Yaskawa INFORM job: aprem2TRJ4.JBI

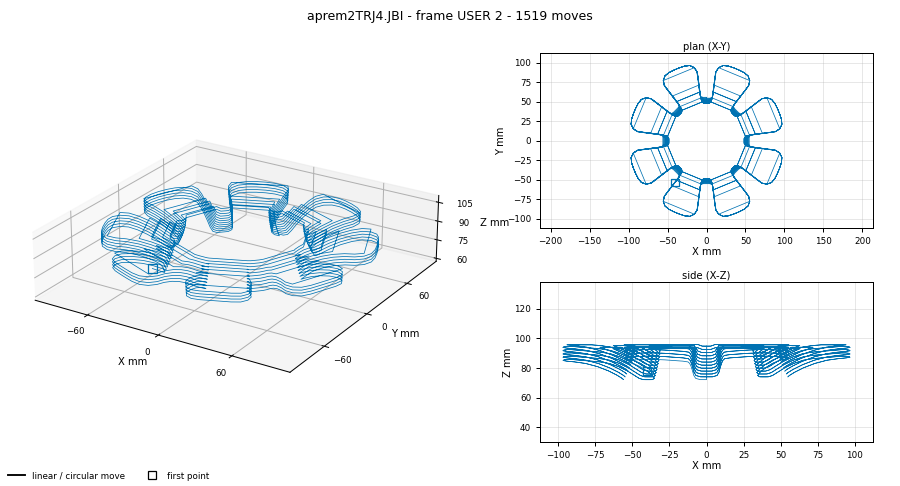
[picture p0: tool path of aprem2TRJ4.JBI in frame USER 2, 1519 of 1519 moves have a stored position in this frame; points joined in program order, loops and branches not executed]
/JOB
//NAME aprem2TRJ4
//POS
///NPOS 1519,0,1519,0,0,0
///USER 2
///TOOL 1
///POSTYPE USER
///RECTAN
///RCONF 1,0,0,0,0,0,0,0,0,0,0,0,0,0,0,0,0,0,0,0,0,0,0,0
C00000=-40.007,-53.324,78.036,177.7295,-3.1005,0.0000
C00001=-36.517,-48.718,75.143,178.8242,-1.7083,0.0000
C00002=-35.037,-45.351,73.015,-179.8825,17.3486,0.0000
C00003=-36.538,-42.505,72.166,160.0580,24.5520,0.0000
C00004=-38.303,-40.803,72.129,156.0408,22.3844,0.0000
C00005=-39.567,-39.567,72.154,156.8171,23.1818,0.0000
C00006=-40.803,-38.303,72.129,157.6162,23.9597,0.0000
C00007=-42.506,-36.538,72.166,155.4471,19.9396,0.0000
C00008=-45.352,-35.037,73.015,162.6519,-0.1179,0.0000
C00009=-48.718,-36.517,75.143,-178.2917,1.1758,0.0000
C00010=-53.324,-40.007,78.036,-176.8995,2.2705,0.0000
C00011=-59.196,-44.618,80.927,-176.4745,2.6327,0.0000
C00012=-65.578,-49.604,83.062,-176.2466,2.8111,0.0000
C00013=-71.524,-53.949,84.088,-176.0077,2.0393,0.0000
C00014=-77.795,-55.184,84.621,-177.1914,-0.2563,0.0000
C00015=-83.601,-53.037,85.050,-178.9039,-0.7847,0.0000
C00016=-87.741,-47.957,85.481,-179.9577,-0.0772,0.0000
C00017=-90.934,-41.602,85.762,-179.9958,-0.0092,0.0000
C00018=-93.717,-34.883,85.762,-179.9965,-0.0095,0.0000
C00019=-95.953,-28.131,85.481,-179.9754,-0.0845,0.0000
C00020=-96.617,-21.612,85.050,179.7797,-1.3299,0.0000
C00021=-94.030,-15.989,84.621,178.1943,-2.1678,0.0000
C00022=-88.723,-12.427,84.088,175.7377,-1.3847,0.0000
C00023=-81.446,-11.295,83.062,175.3629,-0.6685,0.0000
C00024=-73.408,-10.308,80.927,175.6494,-0.6331,0.0000
C00025=-65.995,-9.417,78.036,176.2047,-0.5882,0.0000
C00026=-60.270,-8.627,75.143,177.9610,-0.3768,0.0000
C00027=-56.844,-7.293,73.015,-167.4643,12.3773,0.0000
C00028=-55.892,-4.219,72.166,-176.1973,30.0956,0.0000
C00029=-55.936,-1.768,72.129,178.6826,31.1925,0.0000
C00030=-55.957,0.000,72.154,179.9991,31.1998,0.0000
C00031=-55.936,1.767,72.129,-178.6816,31.1926,0.0000
C00032=-55.892,4.220,72.166,176.1946,30.0948,0.0000
C00033=-56.844,7.293,73.015,167.4645,12.3766,0.0000
C00034=-60.270,8.627,75.143,-177.9610,-0.3768,0.0000
C00035=-65.995,9.417,78.036,-176.2047,-0.5882,0.0000
C00036=-73.408,10.308,80.927,-175.6494,-0.6331,0.0000
C00037=-81.446,11.295,83.062,-175.3629,-0.6685,0.0000
C00038=-88.723,12.427,84.088,-175.7377,-1.3847,0.0000
C00039=-94.030,15.989,84.621,-178.1943,-2.1678,0.0000
C00040=-96.617,21.612,85.050,-179.7797,-1.3299,0.0000
C00041=-95.953,28.131,85.481,179.9754,-0.0845,0.0000
C00042=-93.717,34.883,85.762,179.9965,-0.0095,0.0000
C00043=-90.934,41.602,85.762,179.9958,-0.0092,0.0000
C00044=-87.741,47.957,85.481,179.9577,-0.0772,0.0000
C00045=-83.601,53.037,85.050,178.9039,-0.7847,0.0000
C00046=-77.795,55.184,84.621,177.1914,-0.2563,0.0000
C00047=-71.524,53.949,84.088,176.0077,2.0393,0.0000
C00048=-65.578,49.604,83.062,176.2466,2.8111,0.0000
C00049=-59.196,44.618,80.927,176.4745,2.6327,0.0000
C00050=-53.324,40.007,78.036,176.8995,2.2705,0.0000
C00051=-48.718,36.517,75.143,178.2917,1.1758,0.0000
C00052=-45.351,35.037,73.015,-162.6514,-0.1175,0.0000
C00053=-42.505,36.538,72.166,-155.4480,19.9420,0.0000
C00054=-40.803,38.303,72.129,-157.6156,23.9592,0.0000
C00055=-39.567,39.567,72.154,-156.8182,23.1829,0.0000
C00056=-38.303,40.803,72.129,-156.0403,22.3838,0.0000
C00057=-36.538,42.506,72.166,-160.0604,24.5529,0.0000
C00058=-35.037,45.352,73.015,179.8821,17.3481,0.0000
C00059=-36.517,48.718,75.143,-178.8242,-1.7083,0.0000
C00060=-40.007,53.324,78.036,-177.7295,-3.1005,0.0000
C00061=-44.618,59.196,80.927,-177.3673,-3.5255,0.0000
C00062=-49.604,65.578,83.062,-177.1889,-3.7534,0.0000
C00063=-53.949,71.524,84.088,-177.9607,-3.9923,0.0000
C00064=-55.184,77.795,84.621,179.7437,-2.8086,0.0000
C00065=-53.037,83.601,85.050,179.2153,-1.0961,0.0000
C00066=-47.957,87.741,85.481,179.9228,-0.0423,0.0000
C00067=-41.602,90.934,85.762,179.9908,-0.0042,0.0000
C00068=-34.883,93.717,85.762,179.9905,-0.0035,0.0000
C00069=-28.131,95.953,85.481,179.9155,-0.0246,0.0000
C00070=-21.612,96.617,85.050,178.6701,0.2203,0.0000
C00071=-15.989,94.030,84.621,177.8322,1.8057,0.0000
C00072=-12.427,88.723,84.088,178.6153,4.2623,0.0000
C00073=-11.295,81.446,83.062,179.3315,4.6371,0.0000
C00074=-10.308,73.408,80.927,179.3669,4.3506,0.0000
C00075=-9.417,65.995,78.036,179.4118,3.7953,0.0000
C00076=-8.627,60.270,75.143,179.6232,2.0390,0.0000
C00077=-7.293,56.844,73.015,-167.6234,-12.5355,0.0000
C00078=-4.220,55.892,72.166,-149.9052,-3.8054,0.0000
C00079=-1.767,55.936,72.129,-148.8074,1.3184,0.0000
C00080=0.000,55.957,72.154,-148.8002,-0.0009,0.0000
C00081=0.000,54.840,74.049,-150.2606,-0.0009,0.0000
C00082=1.666,54.823,74.024,-150.2652,-1.1897,0.0000
C00083=4.048,54.790,74.062,-151.4249,3.8705,0.0000
C00084=7.088,55.804,74.943,-168.9167,11.6638,0.0000
C00085=8.393,59.388,77.145,179.6271,-2.1340,0.0000
C00086=9.180,65.335,80.122,179.4707,-3.5331,0.0000
C00087=10.089,72.980,83.074,179.4510,-3.8704,0.0000
C00088=11.094,81.206,85.240,179.4410,-3.9838,0.0000
C00089=12.226,88.613,86.276,178.8532,-3.5972,0.0000
C00090=15.808,94.009,86.813,178.1980,-1.5172,0.0000
C00091=21.475,96.642,87.246,178.9013,-0.1852,0.0000
C00092=28.048,95.980,87.679,179.9308,0.0202,0.0000
C00093=34.856,93.728,87.962,179.9923,0.0029,0.0000
C00094=41.629,90.922,87.962,179.9925,0.0034,0.0000
C00095=48.035,87.701,87.679,179.9368,0.0347,0.0000
C00096=53.151,83.521,87.246,179.3540,0.9079,0.0000
C00097=55.296,77.652,86.813,179.7985,2.3464,0.0000
C00098=54.014,71.304,86.276,-178.2646,3.3541,0.0000
C00099=49.577,65.266,85.240,-177.5752,3.2135,0.0000
C00100=44.470,58.738,83.074,-177.6486,3.1261,0.0000
C00101=39.708,52.690,80.122,-177.8738,2.8733,0.0000
C00102=36.059,47.928,77.145,-178.7542,1.7728,0.0000
C00103=34.447,44.472,74.943,179.5730,-15.8802,0.0000
C00104=35.880,41.605,74.062,-161.3614,-23.4111,0.0000
C00105=37.588,39.944,74.024,-157.2868,-21.2665,0.0000
C00106=38.778,38.778,74.049,-158.0022,-21.9968,0.0000
C00107=39.943,37.588,74.024,-158.7340,-22.7138,0.0000
C00108=41.605,35.880,74.062,-156.5881,-18.6363,0.0000
C00109=44.472,34.447,74.943,-164.1205,0.4274,0.0000
C00110=47.928,36.059,77.145,178.2272,-1.2458,0.0000
C00111=52.690,39.708,80.122,177.1267,-2.1262,0.0000
C00112=58.738,44.470,83.074,176.8739,-2.3514,0.0000
C00113=65.266,49.577,85.240,176.7865,-2.4248,0.0000
C00114=71.304,54.014,86.276,176.6459,-1.7354,0.0000
C00115=77.652,55.296,86.813,177.6536,0.2015,0.0000
C00116=83.521,53.151,87.246,179.0921,0.6460,0.0000
C00117=87.701,48.035,87.679,179.9653,0.0632,0.0000
C00118=90.922,41.629,87.962,179.9966,0.0075,0.0000
C00119=93.728,34.856,87.962,179.9971,0.0077,0.0000
C00120=95.980,28.048,87.679,179.9798,0.0692,0.0000
C00121=96.642,21.475,87.246,-179.8148,1.0987,0.0000
C00122=94.009,15.808,86.813,-178.4828,1.8020,0.0000
C00123=88.613,12.226,86.276,-176.4028,1.1468,0.0000
C00124=81.206,11.094,85.240,-176.0162,0.5590,0.0000
C00125=72.980,10.089,83.074,-176.1296,0.5490,0.0000
C00126=65.335,9.180,80.122,-176.4669,0.5293,0.0000
C00127=59.388,8.393,77.145,-177.8660,0.3729,0.0000
C00128=55.804,7.088,74.943,168.3362,-11.0833,0.0000
C00129=54.790,4.048,74.062,176.1295,-28.5751,0.0000
C00130=54.823,1.666,74.024,-178.8103,-29.7348,0.0000
C00131=54.840,0.000,74.049,-179.9991,-29.7394,0.0000
C00132=54.823,-1.665,74.024,178.8094,-29.7348,0.0000
C00133=54.790,-4.048,74.062,-176.1270,-28.5741,0.0000
C00134=55.804,-7.088,74.943,-168.3364,-11.0826,0.0000
C00135=59.388,-8.393,77.145,177.8660,0.3729,0.0000
C00136=65.335,-9.180,80.122,176.4669,0.5293,0.0000
C00137=72.980,-10.089,83.074,176.1296,0.5490,0.0000
C00138=81.206,-11.094,85.240,176.0162,0.5590,0.0000
C00139=88.613,-12.226,86.276,176.4028,1.1468,0.0000
C00140=94.009,-15.808,86.813,178.4828,1.8020,0.0000
C00141=96.642,-21.475,87.246,179.8148,1.0987,0.0000
C00142=95.980,-28.048,87.679,-179.9798,0.0692,0.0000
C00143=93.728,-34.856,87.962,-179.9971,0.0077,0.0000
C00144=90.922,-41.629,87.962,-179.9966,0.0075,0.0000
C00145=87.701,-48.035,87.679,-179.9653,0.0632,0.0000
C00146=83.521,-53.151,87.246,-179.0921,0.6460,0.0000
C00147=77.652,-55.296,86.813,-177.6536,0.2015,0.0000
C00148=71.304,-54.014,86.276,-176.6459,-1.7354,0.0000
C00149=65.266,-49.577,85.240,-176.7865,-2.4248,0.0000
C00150=58.738,-44.470,83.074,-176.8739,-2.3514,0.0000
C00151=52.690,-39.708,80.122,-177.1267,-2.1262,0.0000
C00152=47.928,-36.059,77.145,-178.2272,-1.2458,0.0000
C00153=44.472,-34.447,74.943,164.1198,0.4270,0.0000
C00154=41.605,-35.880,74.062,156.5889,-18.6386,0.0000
C00155=39.944,-37.588,74.024,158.7335,-22.7132,0.0000
C00156=38.778,-38.778,74.049,158.0032,-21.9978,0.0000
C00157=37.588,-39.943,74.024,157.2862,-21.2660,0.0000
C00158=35.880,-41.605,74.062,161.3637,-23.4119,0.0000
C00159=34.447,-44.472,74.943,-179.5726,-15.8795,0.0000
C00160=36.059,-47.928,77.145,178.7542,1.7728,0.0000
C00161=39.708,-52.690,80.122,177.8738,2.8733,0.0000
C00162=44.470,-58.738,83.074,177.6486,3.1261,0.0000
C00163=49.577,-65.266,85.240,177.5752,3.2135,0.0000
C00164=54.014,-71.304,86.276,178.2646,3.3541,0.0000
C00165=55.296,-77.652,86.813,-179.7985,2.3464,0.0000
C00166=53.151,-83.521,87.246,-179.3540,0.9079,0.0000
C00167=48.035,-87.701,87.679,-179.9368,0.0347,0.0000
C00168=41.629,-90.922,87.962,-179.9925,0.0034,0.0000
C00169=34.856,-93.728,87.962,-179.9923,0.0029,0.0000
C00170=28.048,-95.980,87.679,-179.9308,0.0202,0.0000
C00171=21.475,-96.642,87.246,-178.9013,-0.1852,0.0000
C00172=15.808,-94.009,86.813,-178.1980,-1.5172,0.0000
C00173=12.226,-88.613,86.276,-178.8532,-3.5972,0.0000
C00174=11.094,-81.206,85.240,-179.4410,-3.9838,0.0000
C00175=10.089,-72.980,83.074,-179.4510,-3.8704,0.0000
C00176=9.180,-65.335,80.122,-179.4707,-3.5331,0.0000
C00177=8.393,-59.388,77.145,-179.6271,-2.1340,0.0000
C00178=7.088,-55.804,74.943,168.9167,11.6638,0.0000
C00179=4.048,-54.790,74.062,151.4249,3.8705,0.0000
C00180=1.666,-54.823,74.024,150.2652,-1.1897,0.0000
C00181=0.000,-54.840,74.049,150.2606,-0.0009,0.0000
C00182=0.000,-54.840,74.049,150.2606,-0.0009,0.0000
C00183=-1.665,-54.823,74.024,150.2652,1.1906,0.0000
C00184=-4.048,-54.790,74.062,151.4259,-3.8730,0.0000
C00185=-7.088,-55.804,74.943,168.9174,-11.6636,0.0000
C00186=-8.393,-59.388,77.145,-179.6271,2.1340,0.0000
C00187=-9.180,-65.335,80.122,-179.4707,3.5331,0.0000
C00188=-10.089,-72.980,83.074,-179.4510,3.8704,0.0000
C00189=-11.094,-81.206,85.240,-179.4410,3.9838,0.0000
C00190=-12.226,-88.613,86.276,-178.8532,3.5972,0.0000
C00191=-15.808,-94.009,86.813,-178.1980,1.5172,0.0000
C00192=-21.475,-96.642,87.246,-178.9013,0.1852,0.0000
C00193=-28.048,-95.980,87.679,-179.9308,-0.0202,0.0000
C00194=-34.856,-93.728,87.962,-179.9923,-0.0029,0.0000
C00195=-41.629,-90.922,87.962,-179.9925,-0.0034,0.0000
C00196=-48.035,-87.701,87.679,-179.9368,-0.0347,0.0000
C00197=-53.151,-83.521,87.246,-179.3540,-0.9079,0.0000
C00198=-55.296,-77.652,86.813,-179.7985,-2.3464,0.0000
C00199=-54.014,-71.304,86.276,178.2646,-3.3541,0.0000
C00200=-49.577,-65.266,85.240,177.5752,-3.2135,0.0000
C00201=-44.470,-58.738,83.074,177.6486,-3.1261,0.0000
C00202=-39.708,-52.690,80.122,177.8738,-2.8733,0.0000
C00203=-36.059,-47.928,77.145,178.7542,-1.7728,0.0000
C00204=-34.447,-44.472,74.943,-179.5730,15.8802,0.0000
C00205=-35.880,-41.605,74.062,161.3614,23.4111,0.0000
C00206=-37.588,-39.944,74.024,157.2868,21.2665,0.0000
C00207=-38.778,-38.778,74.049,158.0022,21.9968,0.0000
C00208=-39.943,-37.588,74.024,158.7340,22.7138,0.0000
C00209=-41.605,-35.880,74.062,156.5881,18.6363,0.0000
C00210=-44.472,-34.447,74.943,164.1205,-0.4274,0.0000
C00211=-47.928,-36.059,77.145,-178.2272,1.2458,0.0000
C00212=-52.690,-39.708,80.122,-177.1267,2.1262,0.0000
C00213=-58.738,-44.470,83.074,-176.8739,2.3514,0.0000
C00214=-65.266,-49.577,85.240,-176.7865,2.4248,0.0000
C00215=-71.304,-54.014,86.276,-176.6459,1.7354,0.0000
C00216=-77.652,-55.296,86.813,-177.6536,-0.2015,0.0000
C00217=-83.521,-53.151,87.246,-179.0921,-0.6460,0.0000
C00218=-87.701,-48.035,87.679,-179.9653,-0.0632,0.0000
C00219=-90.922,-41.629,87.962,-179.9966,-0.0075,0.0000
C00220=-93.728,-34.856,87.962,-179.9971,-0.0077,0.0000
C00221=-95.980,-28.048,87.679,-179.9798,-0.0692,0.0000
C00222=-96.642,-21.475,87.246,179.8148,-1.0987,0.0000
C00223=-94.009,-15.808,86.813,178.4828,-1.8020,0.0000
C00224=-88.613,-12.226,86.276,176.4028,-1.1468,0.0000
C00225=-81.206,-11.094,85.240,176.0162,-0.5590,0.0000
C00226=-72.980,-10.089,83.074,176.1296,-0.5490,0.0000
C00227=-65.335,-9.180,80.122,176.4669,-0.5293,0.0000
C00228=-59.388,-8.393,77.145,177.8660,-0.3729,0.0000
C00229=-55.804,-7.088,74.943,-168.3362,11.0833,0.0000
C00230=-54.790,-4.048,74.062,-176.1295,28.5751,0.0000
C00231=-54.823,-1.666,74.024,178.8103,29.7348,0.0000
C00232=-54.840,0.000,74.049,179.9991,29.7394,0.0000
C00233=-54.823,1.665,74.024,-178.8094,29.7348,0.0000
C00234=-54.790,4.048,74.062,176.1270,28.5741,0.0000
C00235=-55.804,7.088,74.943,168.3364,11.0826,0.0000
C00236=-59.388,8.393,77.145,-177.8660,-0.3729,0.0000
C00237=-65.335,9.180,80.122,-176.4669,-0.5293,0.0000
C00238=-72.980,10.089,83.074,-176.1296,-0.5490,0.0000
C00239=-81.206,11.094,85.240,-176.0162,-0.5590,0.0000
C00240=-88.613,12.226,86.276,-176.4028,-1.1468,0.0000
C00241=-94.009,15.808,86.813,-178.4828,-1.8020,0.0000
C00242=-96.642,21.475,87.246,-179.8148,-1.0987,0.0000
C00243=-95.980,28.048,87.679,179.9798,-0.0692,0.0000
C00244=-93.728,34.856,87.962,179.9971,-0.0077,0.0000
C00245=-90.922,41.629,87.962,179.9966,-0.0075,0.0000
C00246=-87.701,48.035,87.679,179.9653,-0.0632,0.0000
C00247=-83.521,53.151,87.246,179.0921,-0.6460,0.0000
C00248=-77.652,55.296,86.813,177.6536,-0.2015,0.0000
C00249=-71.304,54.014,86.276,176.6459,1.7354,0.0000
C00250=-65.266,49.577,85.240,176.7865,2.4248,0.0000
C00251=-58.738,44.470,83.074,176.8739,2.3514,0.0000
C00252=-52.690,39.708,80.122,177.1267,2.1262,0.0000
C00253=-47.928,36.059,77.145,178.2272,1.2458,0.0000
C00254=-44.472,34.447,74.943,-164.1198,-0.4270,0.0000
C00255=-41.605,35.880,74.062,-156.5889,18.6386,0.0000
C00256=-39.944,37.588,74.024,-158.7335,22.7132,0.0000
C00257=-38.778,38.778,74.049,-158.0032,21.9978,0.0000
C00258=-37.588,39.943,74.024,-157.2862,21.2660,0.0000
C00259=-35.880,41.605,74.062,-161.3637,23.4119,0.0000
C00260=-34.447,44.472,74.943,179.5726,15.8795,0.0000
C00261=-36.059,47.928,77.145,-178.7542,-1.7728,0.0000
C00262=-39.708,52.690,80.122,-177.8738,-2.8733,0.0000
C00263=-44.470,58.738,83.074,-177.6486,-3.1261,0.0000
C00264=-49.577,65.266,85.240,-177.5752,-3.2135,0.0000
C00265=-54.014,71.304,86.276,-178.2646,-3.3541,0.0000
C00266=-55.296,77.652,86.813,179.7985,-2.3464,0.0000
C00267=-53.151,83.521,87.246,179.3540,-0.9079,0.0000
C00268=-48.035,87.701,87.679,179.9368,-0.0347,0.0000
C00269=-41.629,90.922,87.962,179.9925,-0.0034,0.0000
C00270=-34.856,93.728,87.962,179.9923,-0.0029,0.0000
C00271=-28.048,95.980,87.679,179.9308,-0.0202,0.0000
C00272=-21.475,96.642,87.246,178.9013,0.1852,0.0000
C00273=-15.808,94.009,86.813,178.1980,1.5172,0.0000
C00274=-12.226,88.613,86.276,178.8532,3.5972,0.0000
C00275=-11.094,81.206,85.240,179.4410,3.9838,0.0000
C00276=-10.089,72.980,83.074,179.4510,3.8704,0.0000
C00277=-9.180,65.335,80.122,179.4707,3.5331,0.0000
C00278=-8.393,59.388,77.145,179.6271,2.1340,0.0000
C00279=-7.088,55.804,74.943,-168.9174,-11.6636,0.0000
C00280=-4.048,54.790,74.062,-151.4259,-3.8730,0.0000
C00281=-1.665,54.823,74.024,-150.2652,1.1906,0.0000
C00282=0.000,54.840,74.049,-150.2606,-0.0009,0.0000
C00283=0.000,53.776,75.975,-151.9017,-0.0008,0.0000
C00284=1.568,53.762,75.948,-151.9034,-1.0593,0.0000
C00285=3.884,53.739,75.988,-153.1148,3.8750,0.0000
C00286=6.894,54.818,76.900,-170.1649,10.7294,0.0000
C00287=8.175,58.565,79.173,179.6434,-2.1517,0.0000
C00288=8.965,64.737,82.228,179.5331,-3.2135,0.0000
C00289=9.898,72.606,85.234,179.5371,-3.3364,0.0000
C00290=10.924,81.005,87.424,179.5509,-3.2738,0.0000
C00291=12.061,88.524,88.468,179.0976,-2.8742,0.0000
C00292=15.662,93.991,89.008,178.5900,-1.1973,0.0000
C00293=21.365,96.662,89.443,179.1515,-0.1450,0.0000
C00294=27.983,96.002,89.878,179.9474,0.0153,0.0000
C00295=34.834,93.736,90.162,179.9942,0.0022,0.0000
C00296=41.650,90.913,90.162,179.9944,0.0026,0.0000
C00297=48.097,87.670,89.878,179.9520,0.0264,0.0000
C00298=53.243,83.458,89.443,179.5025,0.7025,0.0000
C00299=55.387,77.537,89.008,179.8495,1.8433,0.0000
C00300=54.067,71.124,88.468,-178.6043,2.6703,0.0000
C00301=49.554,65.004,87.424,-178.0010,2.6331,0.0000
C00302=44.341,58.339,85.234,-177.9664,2.6872,0.0000
C00303=39.437,52.115,82.228,-178.0562,2.6030,0.0000
C00304=35.631,47.192,79.173,-178.7302,1.7738,0.0000
C00305=33.888,43.637,76.900,179.3468,-14.3899,0.0000
C00306=35.253,40.746,75.988,-162.7447,-22.1169,0.0000
C00307=36.906,39.124,75.948,-158.6653,-20.0234,0.0000
C00308=38.025,38.025,75.975,-159.3164,-20.6826,0.0000
C00309=39.124,36.906,75.948,-159.9771,-21.3352,0.0000
C00310=40.746,35.253,75.988,-157.8823,-17.2529,0.0000
C00311=43.637,33.888,76.901,-165.6107,0.6536,0.0000
C00312=47.192,35.631,79.173,178.2262,-1.2698,0.0000
C00313=52.115,39.437,82.228,177.3970,-1.9438,0.0000
C00314=58.339,44.341,85.234,177.3128,-2.0336,0.0000
C00315=65.004,49.554,87.424,177.3669,-1.9990,0.0000
C00316=71.124,54.067,88.468,177.3297,-1.3957,0.0000
C00317=77.537,55.387,89.008,178.1567,0.1505,0.0000
C00318=83.458,53.243,89.443,179.2975,0.4975,0.0000
C00319=87.670,48.097,89.878,179.9736,0.0480,0.0000
C00320=90.913,41.650,90.162,179.9974,0.0056,0.0000
C00321=93.736,34.834,90.162,179.9978,0.0058,0.0000
C00322=96.002,27.983,89.878,179.9847,0.0526,0.0000
C00323=96.662,21.365,89.443,-179.8550,0.8485,0.0000
C00324=93.991,15.662,89.008,-178.8027,1.4100,0.0000
C00325=88.524,12.061,88.468,-177.1258,0.9024,0.0000
C00326=81.005,10.924,87.424,-176.7262,0.4491,0.0000
C00327=72.606,9.898,85.234,-176.6636,0.4629,0.0000
C00328=64.737,8.965,82.228,-176.7865,0.4669,0.0000
C00329=58.565,8.175,79.173,-177.8483,0.3566,0.0000
C00330=54.818,6.894,76.900,169.2706,-9.8351,0.0000
C00331=53.739,3.884,75.988,176.1250,-26.8852,0.0000
C00332=53.762,1.568,75.948,-178.9407,-28.0966,0.0000
C00333=53.776,0.000,75.975,-179.9992,-28.0983,0.0000
C00334=53.762,-1.568,75.948,178.9399,-28.0967,0.0000
C00335=53.739,-3.885,75.988,-176.1225,-26.8842,0.0000
C00336=54.819,-6.894,76.901,-169.2709,-9.8343,0.0000
C00337=58.565,-8.175,79.173,177.8483,0.3566,0.0000
C00338=64.737,-8.965,82.228,176.7865,0.4669,0.0000
C00339=72.606,-9.898,85.234,176.6636,0.4629,0.0000
C00340=81.005,-10.924,87.424,176.7262,0.4491,0.0000
C00341=88.524,-12.061,88.468,177.1258,0.9024,0.0000
C00342=93.991,-15.662,89.008,178.8027,1.4100,0.0000
C00343=96.662,-21.365,89.443,179.8550,0.8485,0.0000
C00344=96.002,-27.983,89.878,-179.9847,0.0526,0.0000
C00345=93.736,-34.834,90.162,-179.9978,0.0058,0.0000
C00346=90.913,-41.650,90.162,-179.9974,0.0056,0.0000
C00347=87.670,-48.097,89.878,-179.9736,0.0480,0.0000
C00348=83.458,-53.243,89.443,-179.2975,0.4975,0.0000
C00349=77.537,-55.387,89.008,-178.1567,0.1505,0.0000
C00350=71.124,-54.067,88.468,-177.3297,-1.3957,0.0000
C00351=65.004,-49.554,87.424,-177.3669,-1.9990,0.0000
C00352=58.339,-44.341,85.234,-177.3128,-2.0336,0.0000
C00353=52.115,-39.437,82.228,-177.3970,-1.9438,0.0000
C00354=47.192,-35.631,79.173,-178.2262,-1.2698,0.0000
C00355=43.637,-33.888,76.900,165.6101,0.6532,0.0000
C00356=40.746,-35.253,75.988,157.8831,-17.2553,0.0000
C00357=39.124,-36.906,75.948,159.9766,-21.3347,0.0000
C00358=38.025,-38.025,75.975,159.3174,-20.6836,0.0000
C00359=36.906,-39.124,75.948,158.6648,-20.0229,0.0000
C00360=35.253,-40.746,75.988,162.7471,-22.1177,0.0000
C00361=33.888,-43.637,76.901,-179.3464,-14.3893,0.0000
C00362=35.631,-47.192,79.173,178.7302,1.7738,0.0000
C00363=39.437,-52.115,82.228,178.0562,2.6030,0.0000
C00364=44.341,-58.339,85.234,177.9664,2.6872,0.0000
C00365=49.554,-65.004,87.424,178.0010,2.6331,0.0000
C00366=54.067,-71.124,88.468,178.6043,2.6703,0.0000
C00367=55.387,-77.537,89.008,-179.8495,1.8433,0.0000
C00368=53.243,-83.458,89.443,-179.5025,0.7025,0.0000
C00369=48.097,-87.670,89.878,-179.9520,0.0264,0.0000
C00370=41.650,-90.913,90.162,-179.9944,0.0026,0.0000
C00371=34.834,-93.736,90.162,-179.9942,0.0022,0.0000
C00372=27.983,-96.002,89.878,-179.9474,0.0153,0.0000
C00373=21.365,-96.662,89.443,-179.1515,-0.1450,0.0000
C00374=15.662,-93.991,89.008,-178.5900,-1.1973,0.0000
C00375=12.061,-88.524,88.468,-179.0976,-2.8742,0.0000
C00376=10.924,-81.005,87.424,-179.5509,-3.2738,0.0000
C00377=9.898,-72.606,85.234,-179.5371,-3.3364,0.0000
C00378=8.965,-64.737,82.228,-179.5331,-3.2135,0.0000
C00379=8.175,-58.565,79.173,-179.6434,-2.1517,0.0000
C00380=6.894,-54.818,76.900,170.1649,10.7294,0.0000
C00381=3.884,-53.739,75.988,153.1148,3.8750,0.0000
C00382=1.568,-53.762,75.948,151.9034,-1.0593,0.0000
C00383=0.000,-53.776,75.975,151.9017,-0.0008,0.0000
C00384=0.000,-53.776,75.975,151.9017,-0.0008,0.0000
C00385=-1.568,-53.762,75.948,151.9033,1.0601,0.0000
C00386=-3.885,-53.739,75.988,153.1158,-3.8775,0.0000
C00387=-6.894,-54.819,76.901,170.1657,-10.7291,0.0000
C00388=-8.175,-58.565,79.173,-179.6434,2.1517,0.0000
C00389=-8.965,-64.737,82.228,-179.5331,3.2135,0.0000
C00390=-9.898,-72.606,85.234,-179.5371,3.3364,0.0000
C00391=-10.924,-81.005,87.424,-179.5509,3.2738,0.0000
C00392=-12.061,-88.524,88.468,-179.0976,2.8742,0.0000
C00393=-15.662,-93.991,89.008,-178.5900,1.1973,0.0000
C00394=-21.365,-96.662,89.443,-179.1515,0.1450,0.0000
C00395=-27.983,-96.002,89.878,-179.9474,-0.0153,0.0000
C00396=-34.834,-93.736,90.162,-179.9942,-0.0022,0.0000
C00397=-41.650,-90.913,90.162,-179.9944,-0.0026,0.0000
C00398=-48.097,-87.670,89.878,-179.9520,-0.0264,0.0000
C00399=-53.243,-83.458,89.443,-179.5025,-0.7025,0.0000
C00400=-55.387,-77.537,89.008,-179.8495,-1.8433,0.0000
C00401=-54.067,-71.124,88.468,178.6043,-2.6703,0.0000
C00402=-49.554,-65.004,87.424,178.0010,-2.6331,0.0000
C00403=-44.341,-58.339,85.234,177.9664,-2.6872,0.0000
C00404=-39.437,-52.115,82.228,178.0562,-2.6030,0.0000
C00405=-35.631,-47.192,79.173,178.7302,-1.7738,0.0000
C00406=-33.888,-43.637,76.900,-179.3468,14.3899,0.0000
C00407=-35.253,-40.746,75.988,162.7447,22.1169,0.0000
C00408=-36.906,-39.124,75.948,158.6653,20.0234,0.0000
C00409=-38.025,-38.025,75.975,159.3164,20.6826,0.0000
C00410=-39.124,-36.906,75.948,159.9771,21.3352,0.0000
C00411=-40.746,-35.253,75.988,157.8823,17.2529,0.0000
C00412=-43.637,-33.888,76.901,165.6107,-0.6536,0.0000
C00413=-47.192,-35.631,79.173,-178.2262,1.2698,0.0000
C00414=-52.115,-39.437,82.228,-177.3970,1.9438,0.0000
C00415=-58.339,-44.341,85.234,-177.3128,2.0336,0.0000
C00416=-65.004,-49.554,87.424,-177.3669,1.9990,0.0000
C00417=-71.124,-54.067,88.468,-177.3297,1.3957,0.0000
C00418=-77.537,-55.387,89.008,-178.1567,-0.1505,0.0000
C00419=-83.458,-53.243,89.443,-179.2975,-0.4975,0.0000
C00420=-87.670,-48.097,89.878,-179.9736,-0.0480,0.0000
C00421=-90.913,-41.650,90.162,-179.9974,-0.0056,0.0000
C00422=-93.736,-34.834,90.162,-179.9978,-0.0058,0.0000
C00423=-96.002,-27.983,89.878,-179.9847,-0.0526,0.0000
C00424=-96.662,-21.365,89.443,179.8550,-0.8485,0.0000
C00425=-93.991,-15.662,89.008,178.8027,-1.4100,0.0000
C00426=-88.524,-12.061,88.468,177.1258,-0.9024,0.0000
C00427=-81.005,-10.924,87.424,176.7262,-0.4491,0.0000
C00428=-72.606,-9.898,85.234,176.6636,-0.4629,0.0000
C00429=-64.737,-8.965,82.228,176.7865,-0.4669,0.0000
C00430=-58.565,-8.175,79.173,177.8483,-0.3566,0.0000
C00431=-54.818,-6.894,76.900,-169.2706,9.8351,0.0000
C00432=-53.739,-3.884,75.988,-176.1250,26.8852,0.0000
C00433=-53.762,-1.568,75.948,178.9407,28.0966,0.0000
C00434=-53.776,0.000,75.975,179.9992,28.0983,0.0000
C00435=-53.762,1.568,75.948,-178.9399,28.0967,0.0000
C00436=-53.739,3.885,75.988,176.1225,26.8842,0.0000
C00437=-54.819,6.894,76.901,169.2709,9.8343,0.0000
C00438=-58.565,8.175,79.173,-177.8483,-0.3566,0.0000
C00439=-64.737,8.965,82.228,-176.7865,-0.4669,0.0000
C00440=-72.606,9.898,85.234,-176.6636,-0.4629,0.0000
C00441=-81.005,10.924,87.424,-176.7262,-0.4491,0.0000
C00442=-88.524,12.061,88.468,-177.1258,-0.9024,0.0000
C00443=-93.991,15.662,89.008,-178.8027,-1.4100,0.0000
C00444=-96.662,21.365,89.443,-179.8550,-0.8485,0.0000
C00445=-96.002,27.983,89.878,179.9847,-0.0526,0.0000
C00446=-93.736,34.834,90.162,179.9978,-0.0058,0.0000
C00447=-90.913,41.650,90.162,179.9974,-0.0056,0.0000
C00448=-87.670,48.097,89.878,179.9736,-0.0480,0.0000
C00449=-83.458,53.243,89.443,179.2975,-0.4975,0.0000
C00450=-77.537,55.387,89.008,178.1567,-0.1505,0.0000
C00451=-71.124,54.067,88.468,177.3297,1.3957,0.0000
C00452=-65.004,49.554,87.424,177.3669,1.9990,0.0000
C00453=-58.339,44.341,85.234,177.3128,2.0336,0.0000
C00454=-52.115,39.437,82.228,177.3970,1.9438,0.0000
C00455=-47.192,35.631,79.173,178.2262,1.2698,0.0000
C00456=-43.637,33.888,76.900,-165.6101,-0.6532,0.0000
C00457=-40.746,35.253,75.988,-157.8831,17.2553,0.0000
C00458=-39.124,36.906,75.948,-159.9766,21.3347,0.0000
C00459=-38.025,38.025,75.975,-159.3174,20.6836,0.0000
C00460=-36.906,39.124,75.948,-158.6648,20.0229,0.0000
C00461=-35.253,40.746,75.988,-162.7471,22.1177,0.0000
C00462=-33.888,43.637,76.901,179.3464,14.3893,0.0000
C00463=-35.631,47.192,79.173,-178.7302,-1.7738,0.0000
C00464=-39.437,52.115,82.228,-178.0562,-2.6030,0.0000
C00465=-44.341,58.339,85.234,-177.9664,-2.6872,0.0000
C00466=-49.554,65.004,87.424,-178.0010,-2.6331,0.0000
C00467=-54.067,71.124,88.468,-178.6043,-2.6703,0.0000
C00468=-55.387,77.537,89.008,179.8495,-1.8433,0.0000
C00469=-53.243,83.458,89.443,179.5025,-0.7025,0.0000
C00470=-48.097,87.670,89.878,179.9520,-0.0264,0.0000
C00471=-41.650,90.913,90.162,179.9944,-0.0026,0.0000
C00472=-34.834,93.736,90.162,179.9942,-0.0022,0.0000
C00473=-27.983,96.002,89.878,179.9474,-0.0153,0.0000
C00474=-21.365,96.662,89.443,179.1515,0.1450,0.0000
C00475=-15.662,93.991,89.008,178.5900,1.1973,0.0000
C00476=-12.061,88.524,88.468,179.0976,2.8742,0.0000
C00477=-10.924,81.005,87.424,179.5509,3.2738,0.0000
C00478=-9.898,72.606,85.234,179.5371,3.3364,0.0000
C00479=-8.965,64.737,82.228,179.5331,3.2135,0.0000
C00480=-8.175,58.565,79.173,179.6434,2.1517,0.0000
C00481=-6.894,54.819,76.901,-170.1657,-10.7291,0.0000
C00482=-3.885,53.739,75.988,-153.1158,-3.8775,0.0000
C00483=-1.568,53.762,75.948,-151.9033,1.0601,0.0000
C00484=0.000,53.776,75.975,-151.9017,-0.0008,0.0000
C00485=0.000,52.771,77.932,-153.7423,-0.0007,0.0000
C00486=1.476,52.759,77.904,-153.7405,-0.9277,0.0000
C00487=3.730,52.747,77.945,-154.9876,3.8100,0.0000
C00488=6.711,53.894,78.888,-171.3670,9.7384,0.0000
C00489=7.974,57.808,81.229,179.6695,-2.0942,0.0000
C00490=8.774,64.206,84.354,179.5987,-2.8379,0.0000
C00491=9.737,72.291,87.405,179.6254,-2.7503,0.0000
C00492=10.790,80.844,89.614,179.6620,-2.5088,0.0000
C00493=11.935,88.455,90.663,179.3495,-2.0963,0.0000
C00494=15.553,93.978,91.206,179.0073,-0.8482,0.0000
C00495=21.285,96.677,91.642,179.4198,-0.1001,0.0000
C00496=27.936,96.017,92.077,179.9653,0.0101,0.0000
C00497=34.820,93.742,92.362,179.9963,0.0014,0.0000
C00498=41.664,90.907,92.362,179.9964,0.0017,0.0000
C00499=48.140,87.648,92.077,179.9683,0.0174,0.0000
C00500=53.310,83.412,91.642,179.6605,0.4810,0.0000
C00501=55.455,77.451,91.206,179.8978,1.3016,0.0000
C00502=54.108,70.986,90.663,-178.9772,1.9422,0.0000
C00503=49.536,64.795,89.614,-178.4643,2.0133,0.0000
C00504=44.233,58.003,87.405,-178.3191,2.2100,0.0000
C00505=39.197,51.604,84.354,-178.2760,2.2909,0.0000
C00506=35.238,46.514,81.229,-178.7524,1.7146,0.0000
C00507=33.363,42.854,78.888,179.1980,-12.8827,0.0000
C00508=34.660,39.935,77.945,-164.2077,-20.6567,0.0000
C00509=36.262,38.350,77.904,-160.1858,-18.6445,0.0000
C00510=37.314,37.314,77.932,-160.7695,-19.2296,0.0000
C00511=38.350,36.262,77.904,-161.3560,-19.8147,0.0000
C00512=39.935,34.660,77.945,-159.3426,-15.7900,0.0000
C00513=42.854,33.363,78.888,-167.1181,0.8024,0.0000
C00514=46.514,35.238,81.229,178.2854,-1.2476,0.0000
C00515=51.604,39.197,84.354,177.7091,-1.7240,0.0000
C00516=58.003,44.233,87.405,177.7900,-1.6809,0.0000
C00517=64.795,49.536,89.614,177.9867,-1.5357,0.0000
C00518=70.986,54.108,90.663,178.0578,-1.0228,0.0000
C00519=77.451,55.455,91.206,178.6984,0.1022,0.0000
C00520=83.412,53.310,91.642,179.5190,0.3395,0.0000
C00521=87.648,48.140,92.077,179.9826,0.0317,0.0000
C00522=90.907,41.664,92.362,179.9983,0.0036,0.0000
C00523=93.742,34.820,92.362,179.9986,0.0037,0.0000
C00524=96.017,27.936,92.077,179.9899,0.0347,0.0000
C00525=96.677,21.285,91.642,-179.8999,0.5802,0.0000
C00526=93.978,15.553,91.206,-179.1518,0.9927,0.0000
C00527=88.455,11.935,90.663,-177.9037,0.6505,0.0000
C00528=80.844,10.790,89.614,-177.4912,0.3380,0.0000
C00529=72.291,9.737,87.405,-177.2497,0.3746,0.0000
C00530=64.206,8.774,84.354,-177.1621,0.4013,0.0000
C00531=57.808,7.974,81.229,-177.9058,0.3305,0.0000
C00532=53.894,6.711,78.888,170.2616,-8.6330,0.0000
C00533=52.747,3.730,77.945,176.1900,-25.0124,0.0000
C00534=52.759,1.476,77.904,-179.0723,-26.2595,0.0000
C00535=52.771,0.000,77.932,-179.9993,-26.2577,0.0000
C00536=52.759,-1.476,77.904,179.0716,-26.2595,0.0000
C00537=52.747,-3.730,77.945,-176.1877,-25.0114,0.0000
C00538=53.894,-6.711,78.888,-170.2619,-8.6323,0.0000
C00539=57.808,-7.974,81.229,177.9058,0.3305,0.0000
C00540=64.206,-8.774,84.354,177.1621,0.4013,0.0000
C00541=72.291,-9.737,87.405,177.2497,0.3746,0.0000
C00542=80.844,-10.790,89.614,177.4912,0.3380,0.0000
C00543=88.455,-11.935,90.663,177.9037,0.6505,0.0000
C00544=93.978,-15.553,91.206,179.1518,0.9927,0.0000
C00545=96.677,-21.285,91.642,179.8999,0.5802,0.0000
C00546=96.017,-27.936,92.077,-179.9899,0.0347,0.0000
C00547=93.742,-34.820,92.362,-179.9986,0.0037,0.0000
C00548=90.907,-41.664,92.362,-179.9983,0.0036,0.0000
C00549=87.648,-48.140,92.077,-179.9826,0.0317,0.0000
C00550=83.412,-53.310,91.642,-179.5190,0.3395,0.0000
C00551=77.451,-55.455,91.206,-178.6984,0.1022,0.0000
C00552=70.986,-54.108,90.663,-178.0578,-1.0228,0.0000
C00553=64.795,-49.536,89.614,-177.9867,-1.5357,0.0000
C00554=58.003,-44.233,87.405,-177.7900,-1.6809,0.0000
C00555=51.604,-39.197,84.354,-177.7091,-1.7240,0.0000
C00556=46.514,-35.238,81.229,-178.2854,-1.2476,0.0000
C00557=42.854,-33.363,78.888,167.1173,0.8020,0.0000
C00558=39.935,-34.660,77.945,159.3433,-15.7923,0.0000
C00559=38.350,-36.262,77.904,161.3555,-19.8142,0.0000
C00560=37.314,-37.314,77.932,160.7704,-19.2305,0.0000
C00561=36.262,-38.350,77.904,160.1853,-18.6440,0.0000
C00562=34.660,-39.935,77.945,164.2100,-20.6574,0.0000
C00563=33.363,-42.854,78.888,-179.1976,-12.8819,0.0000
C00564=35.238,-46.514,81.229,178.7524,1.7146,0.0000
C00565=39.197,-51.604,84.354,178.2760,2.2909,0.0000
C00566=44.233,-58.003,87.405,178.3191,2.2100,0.0000
C00567=49.536,-64.795,89.614,178.4643,2.0133,0.0000
C00568=54.108,-70.986,90.663,178.9772,1.9422,0.0000
C00569=55.455,-77.451,91.206,-179.8978,1.3016,0.0000
C00570=53.310,-83.412,91.642,-179.6605,0.4810,0.0000
C00571=48.140,-87.648,92.077,-179.9683,0.0174,0.0000
C00572=41.664,-90.907,92.362,-179.9964,0.0017,0.0000
C00573=34.820,-93.742,92.362,-179.9963,0.0014,0.0000
C00574=27.936,-96.017,92.077,-179.9653,0.0101,0.0000
C00575=21.285,-96.677,91.642,-179.4198,-0.1001,0.0000
C00576=15.553,-93.978,91.206,-179.0073,-0.8482,0.0000
C00577=11.935,-88.455,90.663,-179.3495,-2.0963,0.0000
C00578=10.790,-80.844,89.614,-179.6620,-2.5088,0.0000
C00579=9.737,-72.291,87.405,-179.6254,-2.7503,0.0000
C00580=8.774,-64.206,84.354,-179.5987,-2.8379,0.0000
C00581=7.974,-57.808,81.229,-179.6695,-2.0942,0.0000
C00582=6.711,-53.894,78.888,171.3670,9.7384,0.0000
C00583=3.730,-52.747,77.945,154.9876,3.8100,0.0000
C00584=1.476,-52.759,77.904,153.7405,-0.9277,0.0000
C00585=0.000,-52.771,77.932,153.7423,-0.0007,0.0000
C00586=0.000,-52.771,77.932,153.7423,-0.0007,0.0000
C00587=-1.476,-52.759,77.904,153.7405,0.9284,0.0000
C00588=-3.730,-52.747,77.945,154.9886,-3.8123,0.0000
C00589=-6.711,-53.894,78.888,171.3677,-9.7381,0.0000
C00590=-7.974,-57.808,81.229,-179.6695,2.0942,0.0000
C00591=-8.774,-64.206,84.354,-179.5987,2.8379,0.0000
C00592=-9.737,-72.291,87.405,-179.6254,2.7503,0.0000
C00593=-10.790,-80.844,89.614,-179.6620,2.5088,0.0000
C00594=-11.935,-88.455,90.663,-179.3495,2.0963,0.0000
C00595=-15.553,-93.978,91.206,-179.0073,0.8482,0.0000
C00596=-21.285,-96.677,91.642,-179.4198,0.1001,0.0000
C00597=-27.936,-96.017,92.077,-179.9653,-0.0101,0.0000
C00598=-34.820,-93.742,92.362,-179.9963,-0.0014,0.0000
C00599=-41.664,-90.907,92.362,-179.9964,-0.0017,0.0000
C00600=-48.140,-87.648,92.077,-179.9683,-0.0174,0.0000
C00601=-53.310,-83.412,91.642,-179.6605,-0.4810,0.0000
C00602=-55.455,-77.451,91.206,-179.8978,-1.3016,0.0000
C00603=-54.108,-70.986,90.663,178.9772,-1.9422,0.0000
C00604=-49.536,-64.795,89.614,178.4643,-2.0133,0.0000
C00605=-44.233,-58.003,87.405,178.3191,-2.2100,0.0000
C00606=-39.197,-51.604,84.354,178.2760,-2.2909,0.0000
C00607=-35.238,-46.514,81.229,178.7524,-1.7146,0.0000
C00608=-33.363,-42.854,78.888,-179.1980,12.8827,0.0000
C00609=-34.660,-39.935,77.945,164.2077,20.6567,0.0000
C00610=-36.262,-38.350,77.904,160.1858,18.6445,0.0000
C00611=-37.314,-37.314,77.932,160.7695,19.2296,0.0000
C00612=-38.350,-36.262,77.904,161.3560,19.8147,0.0000
C00613=-39.935,-34.660,77.945,159.3426,15.7900,0.0000
C00614=-42.854,-33.363,78.888,167.1181,-0.8024,0.0000
C00615=-46.514,-35.238,81.229,-178.2854,1.2476,0.0000
C00616=-51.604,-39.197,84.354,-177.7091,1.7240,0.0000
C00617=-58.003,-44.233,87.405,-177.7900,1.6809,0.0000
C00618=-64.795,-49.536,89.614,-177.9867,1.5357,0.0000
C00619=-70.986,-54.108,90.663,-178.0578,1.0228,0.0000
C00620=-77.451,-55.455,91.206,-178.6984,-0.1022,0.0000
C00621=-83.412,-53.310,91.642,-179.5190,-0.3395,0.0000
C00622=-87.648,-48.140,92.077,-179.9826,-0.0317,0.0000
C00623=-90.907,-41.664,92.362,-179.9983,-0.0036,0.0000
C00624=-93.742,-34.820,92.362,-179.9986,-0.0037,0.0000
C00625=-96.017,-27.936,92.077,-179.9899,-0.0347,0.0000
C00626=-96.677,-21.285,91.642,179.8999,-0.5802,0.0000
C00627=-93.978,-15.553,91.206,179.1518,-0.9927,0.0000
C00628=-88.455,-11.935,90.663,177.9037,-0.6505,0.0000
C00629=-80.844,-10.790,89.614,177.4912,-0.3380,0.0000
C00630=-72.291,-9.737,87.405,177.2497,-0.3746,0.0000
C00631=-64.206,-8.774,84.354,177.1621,-0.4013,0.0000
C00632=-57.808,-7.974,81.229,177.9058,-0.3305,0.0000
C00633=-53.894,-6.711,78.888,-170.2616,8.6330,0.0000
C00634=-52.747,-3.730,77.945,-176.1900,25.0124,0.0000
C00635=-52.759,-1.476,77.904,179.0723,26.2595,0.0000
C00636=-52.771,0.000,77.932,179.9993,26.2577,0.0000
C00637=-52.759,1.476,77.904,-179.0716,26.2595,0.0000
C00638=-52.747,3.730,77.945,176.1877,25.0114,0.0000
C00639=-53.894,6.711,78.888,170.2619,8.6323,0.0000
C00640=-57.808,7.974,81.229,-177.9058,-0.3305,0.0000
C00641=-64.206,8.774,84.354,-177.1621,-0.4013,0.0000
C00642=-72.291,9.737,87.405,-177.2497,-0.3746,0.0000
C00643=-80.844,10.790,89.614,-177.4912,-0.3380,0.0000
C00644=-88.455,11.935,90.663,-177.9037,-0.6505,0.0000
C00645=-93.978,15.553,91.206,-179.1518,-0.9927,0.0000
C00646=-96.677,21.285,91.642,-179.8999,-0.5802,0.0000
C00647=-96.017,27.936,92.077,179.9899,-0.0347,0.0000
C00648=-93.742,34.820,92.362,179.9986,-0.0037,0.0000
C00649=-90.907,41.664,92.362,179.9983,-0.0036,0.0000
C00650=-87.648,48.140,92.077,179.9826,-0.0317,0.0000
C00651=-83.412,53.310,91.642,179.5190,-0.3395,0.0000
C00652=-77.451,55.455,91.206,178.6984,-0.1022,0.0000
C00653=-70.986,54.108,90.663,178.0578,1.0228,0.0000
C00654=-64.795,49.536,89.614,177.9867,1.5357,0.0000
C00655=-58.003,44.233,87.405,177.7900,1.6809,0.0000
C00656=-51.604,39.197,84.354,177.7091,1.7240,0.0000
C00657=-46.514,35.238,81.229,178.2854,1.2476,0.0000
C00658=-42.854,33.363,78.888,-167.1173,-0.8020,0.0000
C00659=-39.935,34.660,77.945,-159.3433,15.7923,0.0000
C00660=-38.350,36.262,77.904,-161.3555,19.8142,0.0000
C00661=-37.314,37.314,77.932,-160.7704,19.2305,0.0000
C00662=-36.262,38.350,77.904,-160.1853,18.6440,0.0000
C00663=-34.660,39.935,77.945,-164.2100,20.6574,0.0000
C00664=-33.363,42.854,78.888,179.1976,12.8819,0.0000
C00665=-35.238,46.514,81.229,-178.7524,-1.7146,0.0000
C00666=-39.197,51.604,84.354,-178.2760,-2.2909,0.0000
C00667=-44.233,58.003,87.405,-178.3191,-2.2100,0.0000
C00668=-49.536,64.795,89.614,-178.4643,-2.0133,0.0000
C00669=-54.108,70.986,90.663,-178.9772,-1.9422,0.0000
C00670=-55.455,77.451,91.206,179.8978,-1.3016,0.0000
C00671=-53.310,83.412,91.642,179.6605,-0.4810,0.0000
C00672=-48.140,87.648,92.077,179.9683,-0.0174,0.0000
C00673=-41.664,90.907,92.362,179.9964,-0.0017,0.0000
C00674=-34.820,93.742,92.362,179.9963,-0.0014,0.0000
C00675=-27.936,96.017,92.077,179.9653,-0.0101,0.0000
C00676=-21.285,96.677,91.642,179.4198,0.1001,0.0000
C00677=-15.553,93.978,91.206,179.0073,0.8482,0.0000
C00678=-11.935,88.455,90.663,179.3495,2.0963,0.0000
C00679=-10.790,80.844,89.614,179.6620,2.5088,0.0000
C00680=-9.737,72.291,87.405,179.6254,2.7503,0.0000
C00681=-8.774,64.206,84.354,179.5987,2.8379,0.0000
C00682=-7.974,57.808,81.229,179.6695,2.0942,0.0000
C00683=-6.711,53.894,78.888,-171.3677,-9.7381,0.0000
C00684=-3.730,52.747,77.945,-154.9886,-3.8123,0.0000
C00685=-1.476,52.759,77.904,-153.7405,0.9284,0.0000
C00686=0.000,52.771,77.932,-153.7423,-0.0007,0.0000
C00687=0.000,51.832,79.921,-155.8023,-0.0006,0.0000
C00688=1.391,51.822,79.893,-155.7966,-0.7969,0.0000
C00689=3.586,51.820,79.935,-157.0572,3.6693,0.0000
C00690=6.543,53.038,80.908,-172.5244,8.6955,0.0000
C00691=7.793,57.125,83.313,179.7036,-1.9641,0.0000
C00692=8.610,63.749,86.500,179.6672,-2.4084,0.0000
C00693=9.608,72.041,89.587,179.7163,-2.1143,0.0000
C00694=10.692,80.728,91.809,179.7750,-1.6915,0.0000
C00695=11.850,88.408,92.861,179.6101,-1.2664,0.0000
C00696=15.484,93.970,93.405,179.4490,-0.4726,0.0000
C00697=21.237,96.685,93.841,179.7050,-0.0512,0.0000
C00698=27.910,96.026,94.277,179.9843,0.0045,0.0000
C00699=34.811,93.745,94.562,179.9985,0.0006,0.0000
C00700=41.672,90.903,94.562,179.9985,0.0007,0.0000
C00701=48.166,87.636,94.277,179.9857,0.0079,0.0000
C00702=53.350,83.383,93.841,179.8276,0.2448,0.0000
C00703=55.498,77.395,93.405,179.9446,0.7238,0.0000
C00704=54.135,70.893,92.861,-179.3801,1.1712,0.0000
C00705=49.523,64.644,91.809,-178.9628,1.3552,0.0000
C00706=44.146,57.735,89.587,-178.7052,1.6958,0.0000
C00707=38.990,51.166,86.500,-178.5316,1.9386,0.0000
C00708=34.883,45.903,83.313,-178.8204,1.5986,0.0000
C00709=32.877,42.130,80.908,179.1200,-11.3613,0.0000
C00710=34.107,39.178,79.935,-165.7499,-19.0172,0.0000
C00711=35.661,37.627,79.893,-161.8574,-17.1189,0.0000
C00712=36.651,36.651,79.921,-162.3718,-17.6274,0.0000
C00713=37.627,35.661,79.893,-162.8815,-18.1429,0.0000
C00714=39.178,34.107,79.935,-160.9822,-14.2479,0.0000
C00715=42.130,32.877,80.908,-168.6394,0.8803,0.0000
C00716=45.903,34.883,83.313,178.4014,-1.1796,0.0000
C00717=51.166,38.990,86.500,178.0614,-1.4684,0.0000
C00718=57.735,44.146,89.587,178.3042,-1.2948,0.0000
C00719=64.644,49.523,91.809,178.6448,-1.0372,0.0000
C00720=70.893,54.135,92.861,178.8288,-0.6199,0.0000
C00721=77.395,55.498,93.405,179.2762,0.0554,0.0000
C00722=83.383,53.350,93.841,179.7552,0.1724,0.0000
C00723=87.636,48.166,94.277,179.9921,0.0143,0.0000
C00724=90.903,41.672,94.562,179.9993,0.0015,0.0000
C00725=93.745,34.811,94.562,179.9994,0.0015,0.0000
C00726=96.026,27.910,94.277,179.9955,0.0157,0.0000
C00727=96.685,21.237,93.841,-179.9488,0.2950,0.0000
C00728=93.970,15.484,93.405,-179.5274,0.5510,0.0000
C00729=88.408,11.850,92.861,-178.7336,0.3899,0.0000
C00730=80.728,10.692,91.809,-178.3085,0.2250,0.0000
C00731=72.041,9.608,89.587,-177.8857,0.2837,0.0000
C00732=63.749,8.610,86.500,-177.5916,0.3328,0.0000
C00733=57.125,7.793,83.313,-178.0359,0.2964,0.0000
C00734=53.038,6.543,80.908,171.3045,-7.4756,0.0000
C00735=51.820,3.586,79.935,176.3307,-22.9428,0.0000
C00736=51.822,1.391,79.893,-179.2031,-24.2034,0.0000
C00737=51.832,0.000,79.921,-179.9994,-24.1977,0.0000
C00738=51.822,-1.390,79.893,179.2025,-24.2034,0.0000
C00739=51.820,-3.586,79.935,-176.3285,-22.9418,0.0000
C00740=53.038,-6.543,80.908,-171.3048,-7.4749,0.0000
C00741=57.125,-7.793,83.313,178.0359,0.2964,0.0000
C00742=63.749,-8.610,86.500,177.5916,0.3328,0.0000
C00743=72.041,-9.608,89.587,177.8857,0.2837,0.0000
C00744=80.728,-10.692,91.809,178.3085,0.2250,0.0000
C00745=88.408,-11.850,92.861,178.7336,0.3899,0.0000
C00746=93.970,-15.484,93.405,179.5274,0.5510,0.0000
C00747=96.685,-21.237,93.841,179.9488,0.2950,0.0000
C00748=96.026,-27.910,94.277,-179.9955,0.0157,0.0000
C00749=93.745,-34.811,94.562,-179.9994,0.0015,0.0000
C00750=90.903,-41.672,94.562,-179.9993,0.0015,0.0000
C00751=87.636,-48.166,94.277,-179.9921,0.0143,0.0000
C00752=83.383,-53.350,93.841,-179.7552,0.1724,0.0000
C00753=77.395,-55.498,93.405,-179.2762,0.0554,0.0000
C00754=70.893,-54.135,92.861,-178.8288,-0.6199,0.0000
C00755=64.644,-49.523,91.809,-178.6448,-1.0372,0.0000
C00756=57.735,-44.146,89.587,-178.3042,-1.2948,0.0000
C00757=51.166,-38.990,86.500,-178.0614,-1.4684,0.0000
C00758=45.903,-34.883,83.313,-178.4014,-1.1796,0.0000
C00759=42.130,-32.877,80.908,168.6387,0.8800,0.0000
C00760=39.178,-34.107,79.935,160.9828,-14.2501,0.0000
C00761=37.627,-35.661,79.893,162.8811,-18.1426,0.0000
C00762=36.651,-36.651,79.921,162.3726,-17.6282,0.0000
C00763=35.661,-37.627,79.893,161.8571,-17.1185,0.0000
C00764=34.107,-39.178,79.935,165.7521,-19.0178,0.0000
C00765=32.877,-42.130,80.908,-179.1197,-11.3606,0.0000
C00766=34.883,-45.903,83.313,178.8204,1.5986,0.0000
C00767=38.990,-51.166,86.500,178.5316,1.9386,0.0000
C00768=44.146,-57.735,89.587,178.7052,1.6958,0.0000
C00769=49.523,-64.644,91.809,178.9628,1.3552,0.0000
C00770=54.135,-70.893,92.861,179.3801,1.1712,0.0000
C00771=55.498,-77.395,93.405,-179.9446,0.7238,0.0000
C00772=53.350,-83.383,93.841,-179.8276,0.2448,0.0000
C00773=48.166,-87.636,94.277,-179.9857,0.0079,0.0000
C00774=41.672,-90.903,94.562,-179.9985,0.0007,0.0000
C00775=34.811,-93.745,94.562,-179.9985,0.0006,0.0000
C00776=27.910,-96.026,94.277,-179.9843,0.0045,0.0000
C00777=21.237,-96.685,93.841,-179.7050,-0.0512,0.0000
C00778=15.484,-93.970,93.405,-179.4490,-0.4726,0.0000
C00779=11.850,-88.408,92.861,-179.6101,-1.2664,0.0000
C00780=10.692,-80.728,91.809,-179.7750,-1.6915,0.0000
C00781=9.608,-72.041,89.587,-179.7163,-2.1143,0.0000
C00782=8.610,-63.749,86.500,-179.6672,-2.4084,0.0000
C00783=7.793,-57.125,83.313,-179.7036,-1.9641,0.0000
C00784=6.543,-53.038,80.908,172.5244,8.6955,0.0000
C00785=3.586,-51.820,79.935,157.0572,3.6693,0.0000
C00786=1.391,-51.822,79.893,155.7966,-0.7969,0.0000
C00787=0.000,-51.832,79.921,155.8023,-0.0006,0.0000
C00788=0.000,-51.832,79.921,155.8023,-0.0006,0.0000
C00789=-1.390,-51.822,79.893,155.7966,0.7975,0.0000
C00790=-3.586,-51.820,79.935,157.0582,-3.6715,0.0000
C00791=-6.543,-53.038,80.908,172.5251,-8.6952,0.0000
C00792=-7.793,-57.125,83.313,-179.7036,1.9641,0.0000
C00793=-8.610,-63.749,86.500,-179.6672,2.4084,0.0000
C00794=-9.608,-72.041,89.587,-179.7163,2.1143,0.0000
C00795=-10.692,-80.728,91.809,-179.7750,1.6915,0.0000
C00796=-11.850,-88.408,92.861,-179.6101,1.2664,0.0000
C00797=-15.484,-93.970,93.405,-179.4490,0.4726,0.0000
C00798=-21.237,-96.685,93.841,-179.7050,0.0512,0.0000
C00799=-27.910,-96.026,94.277,-179.9843,-0.0045,0.0000
C00800=-34.811,-93.745,94.562,-179.9985,-0.0006,0.0000
C00801=-41.672,-90.903,94.562,-179.9985,-0.0007,0.0000
C00802=-48.166,-87.636,94.277,-179.9857,-0.0079,0.0000
C00803=-53.350,-83.383,93.841,-179.8276,-0.2448,0.0000
C00804=-55.498,-77.395,93.405,-179.9446,-0.7238,0.0000
C00805=-54.135,-70.893,92.861,179.3801,-1.1712,0.0000
C00806=-49.523,-64.644,91.809,178.9628,-1.3552,0.0000
C00807=-44.146,-57.735,89.587,178.7052,-1.6958,0.0000
C00808=-38.990,-51.166,86.500,178.5316,-1.9386,0.0000
C00809=-34.883,-45.903,83.313,178.8204,-1.5986,0.0000
C00810=-32.877,-42.130,80.908,-179.1200,11.3613,0.0000
C00811=-34.107,-39.178,79.935,165.7499,19.0172,0.0000
C00812=-35.661,-37.627,79.893,161.8574,17.1189,0.0000
C00813=-36.651,-36.651,79.921,162.3718,17.6274,0.0000
C00814=-37.627,-35.661,79.893,162.8815,18.1429,0.0000
C00815=-39.178,-34.107,79.935,160.9822,14.2479,0.0000
C00816=-42.130,-32.877,80.908,168.6394,-0.8803,0.0000
C00817=-45.903,-34.883,83.313,-178.4014,1.1796,0.0000
C00818=-51.166,-38.990,86.500,-178.0614,1.4684,0.0000
C00819=-57.735,-44.146,89.587,-178.3042,1.2948,0.0000
C00820=-64.644,-49.523,91.809,-178.6448,1.0372,0.0000
C00821=-70.893,-54.135,92.861,-178.8288,0.6199,0.0000
C00822=-77.395,-55.498,93.405,-179.2762,-0.0554,0.0000
C00823=-83.383,-53.350,93.841,-179.7552,-0.1724,0.0000
C00824=-87.636,-48.166,94.277,-179.9921,-0.0143,0.0000
C00825=-90.903,-41.672,94.562,-179.9993,-0.0015,0.0000
C00826=-93.745,-34.811,94.562,-179.9994,-0.0015,0.0000
C00827=-96.026,-27.910,94.277,-179.9955,-0.0157,0.0000
C00828=-96.685,-21.237,93.841,179.9488,-0.2950,0.0000
C00829=-93.970,-15.484,93.405,179.5274,-0.5510,0.0000
C00830=-88.408,-11.850,92.861,178.7336,-0.3899,0.0000
C00831=-80.728,-10.692,91.809,178.3085,-0.2250,0.0000
C00832=-72.041,-9.608,89.587,177.8857,-0.2837,0.0000
C00833=-63.749,-8.610,86.500,177.5916,-0.3328,0.0000
C00834=-57.125,-7.793,83.313,178.0359,-0.2964,0.0000
C00835=-53.038,-6.543,80.908,-171.3045,7.4756,0.0000
C00836=-51.820,-3.586,79.935,-176.3307,22.9428,0.0000
C00837=-51.822,-1.391,79.893,179.2031,24.2034,0.0000
C00838=-51.832,0.000,79.921,179.9994,24.1977,0.0000
C00839=-51.822,1.390,79.893,-179.2025,24.2034,0.0000
C00840=-51.820,3.586,79.935,176.3285,22.9418,0.0000
C00841=-53.038,6.543,80.908,171.3048,7.4749,0.0000
C00842=-57.125,7.793,83.313,-178.0359,-0.2964,0.0000
C00843=-63.749,8.610,86.500,-177.5916,-0.3328,0.0000
C00844=-72.041,9.608,89.587,-177.8857,-0.2837,0.0000
C00845=-80.728,10.692,91.809,-178.3085,-0.2250,0.0000
C00846=-88.408,11.850,92.861,-178.7336,-0.3899,0.0000
C00847=-93.970,15.484,93.405,-179.5274,-0.5510,0.0000
C00848=-96.685,21.237,93.841,-179.9488,-0.2950,0.0000
C00849=-96.026,27.910,94.277,179.9955,-0.0157,0.0000
C00850=-93.745,34.811,94.562,179.9994,-0.0015,0.0000
C00851=-90.903,41.672,94.562,179.9993,-0.0015,0.0000
C00852=-87.636,48.166,94.277,179.9921,-0.0143,0.0000
C00853=-83.383,53.350,93.841,179.7552,-0.1724,0.0000
C00854=-77.395,55.498,93.405,179.2762,-0.0554,0.0000
C00855=-70.893,54.135,92.861,178.8288,0.6199,0.0000
C00856=-64.644,49.523,91.809,178.6448,1.0372,0.0000
C00857=-57.735,44.146,89.587,178.3042,1.2948,0.0000
C00858=-51.166,38.990,86.500,178.0614,1.4684,0.0000
C00859=-45.903,34.883,83.313,178.4014,1.1796,0.0000
C00860=-42.130,32.877,80.908,-168.6387,-0.8800,0.0000
C00861=-39.178,34.107,79.935,-160.9828,14.2501,0.0000
C00862=-37.627,35.661,79.893,-162.8811,18.1426,0.0000
C00863=-36.651,36.651,79.921,-162.3726,17.6282,0.0000
C00864=-35.661,37.627,79.893,-161.8571,17.1185,0.0000
C00865=-34.107,39.178,79.935,-165.7521,19.0178,0.0000
C00866=-32.877,42.130,80.908,179.1197,11.3606,0.0000
C00867=-34.883,45.903,83.313,-178.8204,-1.5986,0.0000
C00868=-38.990,51.166,86.500,-178.5316,-1.9386,0.0000
C00869=-44.146,57.735,89.587,-178.7052,-1.6958,0.0000
C00870=-49.523,64.644,91.809,-178.9628,-1.3552,0.0000
C00871=-54.135,70.893,92.861,-179.3801,-1.1712,0.0000
C00872=-55.498,77.395,93.405,179.9446,-0.7238,0.0000
C00873=-53.350,83.383,93.841,179.8276,-0.2448,0.0000
C00874=-48.166,87.636,94.277,179.9857,-0.0079,0.0000
C00875=-41.672,90.903,94.562,179.9985,-0.0007,0.0000
C00876=-34.811,93.745,94.562,179.9985,-0.0006,0.0000
C00877=-27.910,96.026,94.277,179.9843,-0.0045,0.0000
C00878=-21.237,96.685,93.841,179.7050,0.0512,0.0000
C00879=-15.484,93.970,93.405,179.4490,0.4726,0.0000
C00880=-11.850,88.408,92.861,179.6101,1.2664,0.0000
C00881=-10.692,80.728,91.809,179.7750,1.6915,0.0000
C00882=-9.608,72.041,89.587,179.7163,2.1143,0.0000
C00883=-8.610,63.749,86.500,179.6672,2.4084,0.0000
C00884=-7.793,57.125,83.313,179.7036,1.9641,0.0000
C00885=-6.543,53.038,80.908,-172.5251,-8.6952,0.0000
C00886=-3.586,51.820,79.935,-157.0582,-3.6715,0.0000
C00887=-1.390,51.822,79.893,-155.7966,0.7975,0.0000
C00888=0.000,51.832,79.921,-155.8023,-0.0006,0.0000
C00889=0.000,50.970,81.946,-158.1022,-0.0005,0.0000
C00890=1.312,50.962,81.916,-158.0920,-0.6690,0.0000
C00891=3.453,50.970,81.960,-159.3373,3.4481,0.0000
C00892=6.389,52.261,82.960,-173.6406,7.6045,0.0000
C00893=7.633,56.525,85.423,179.7440,-1.7649,0.0000
C00894=8.475,63.374,88.663,179.7387,-1.9278,0.0000
C00895=9.515,71.858,91.777,179.8100,-1.4311,0.0000
C00896=10.634,80.658,94.007,179.8912,-0.8247,0.0000
C00897=11.808,88.386,95.061,179.8809,-0.3884,0.0000
C00898=15.455,93.966,95.604,179.9140,-0.0739,0.0000
C00899=55.516,77.372,95.604,179.9914,0.1131,0.0000
C00900=54.149,70.847,95.061,-179.8096,0.3589,0.0000
C00901=49.515,64.553,94.007,-179.4937,0.6602,0.0000
C00902=44.083,57.539,91.777,-179.1223,1.1463,0.0000
C00903=38.820,50.805,88.663,-178.8213,1.5481,0.0000
C00904=34.571,45.367,85.423,-178.9328,1.4291,0.0000
C00905=32.436,41.472,82.960,179.1064,-9.8268,0.0000
C00906=33.599,38.483,81.960,-167.3708,-17.1854,0.0000
C00907=35.108,36.963,81.916,-163.6891,-15.4355,0.0000
C00908=36.041,36.041,81.946,-164.1333,-15.8661,0.0000
C00909=36.963,35.108,81.916,-164.5648,-16.3112,0.0000
C00910=38.483,33.599,81.960,-162.8140,-12.6271,0.0000
C00911=41.472,32.436,82.960,-170.1739,0.8939,0.0000
C00912=45.367,34.571,85.423,178.5709,-1.0672,0.0000
C00913=50.805,38.820,88.663,178.4519,-1.1787,0.0000
C00914=57.539,44.083,91.777,178.8537,-0.8777,0.0000
C00915=64.553,49.515,94.007,179.3398,-0.5063,0.0000
C00916=70.847,54.149,95.061,179.6411,-0.1904,0.0000
C00917=77.372,55.516,95.604,179.8869,0.0086,0.0000
C00918=93.966,15.455,95.604,-179.9261,0.0860,0.0000
C00919=88.386,11.808,95.061,-179.6116,0.1191,0.0000
C00920=80.658,10.634,94.007,-179.1753,0.1088,0.0000
C00921=71.858,9.515,91.777,-178.5689,0.1900,0.0000
C00922=63.374,8.475,88.663,-178.0722,0.2613,0.0000
C00923=56.525,7.633,85.423,-178.2351,0.2560,0.0000
C00924=52.261,6.389,82.960,172.3955,-6.3594,0.0000
C00925=50.970,3.453,81.960,176.5519,-20.6627,0.0000
C00926=50.962,1.312,81.916,-179.3310,-21.9080,0.0000
C00927=50.970,0.000,81.946,-179.9995,-21.8978,0.0000
C00928=50.962,-1.311,81.916,179.3306,-21.9080,0.0000
C00929=50.970,-3.454,81.960,-176.5499,-20.6618,0.0000
C00930=52.261,-6.389,82.960,-172.3958,-6.3587,0.0000
C00931=56.525,-7.633,85.423,178.2351,0.2560,0.0000
C00932=63.374,-8.475,88.663,178.0722,0.2613,0.0000
C00933=71.858,-9.515,91.777,178.5689,0.1900,0.0000
C00934=80.658,-10.634,94.007,179.1753,0.1088,0.0000
C00935=88.386,-11.808,95.061,179.6116,0.1191,0.0000
C00936=93.966,-15.455,95.604,179.9261,0.0860,0.0000
C00937=77.372,-55.516,95.604,-179.8869,0.0086,0.0000
C00938=70.847,-54.149,95.061,-179.6411,-0.1904,0.0000
C00939=64.553,-49.515,94.007,-179.3398,-0.5063,0.0000
C00940=57.539,-44.083,91.777,-178.8537,-0.8777,0.0000
C00941=50.805,-38.820,88.663,-178.4519,-1.1787,0.0000
C00942=45.367,-34.571,85.423,-178.5709,-1.0672,0.0000
C00943=41.472,-32.436,82.960,170.1732,0.8936,0.0000
C00944=38.483,-33.599,81.960,162.8146,-12.6292,0.0000
C00945=36.963,-35.108,81.916,164.5645,-16.3109,0.0000
C00946=36.041,-36.041,81.946,164.1339,-15.8667,0.0000
C00947=35.108,-36.963,81.916,163.6888,-15.4352,0.0000
C00948=33.599,-38.483,81.960,167.3729,-17.1860,0.0000
C00949=32.436,-41.472,82.960,-179.1061,-9.8261,0.0000
C00950=34.571,-45.367,85.423,178.9328,1.4291,0.0000
C00951=38.820,-50.805,88.663,178.8213,1.5481,0.0000
C00952=44.083,-57.539,91.777,179.1223,1.1463,0.0000
C00953=49.515,-64.553,94.007,179.4937,0.6602,0.0000
C00954=54.149,-70.847,95.061,179.8096,0.3589,0.0000
C00955=55.516,-77.372,95.604,-179.9914,0.1131,0.0000
C00956=15.455,-93.966,95.604,-179.9140,-0.0739,0.0000
C00957=11.808,-88.386,95.061,-179.8809,-0.3884,0.0000
C00958=10.634,-80.658,94.007,-179.8912,-0.8247,0.0000
C00959=9.515,-71.858,91.777,-179.8100,-1.4311,0.0000
C00960=8.475,-63.374,88.663,-179.7387,-1.9278,0.0000
C00961=7.633,-56.525,85.423,-179.7440,-1.7649,0.0000
C00962=6.389,-52.261,82.960,173.6406,7.6045,0.0000
C00963=3.453,-50.970,81.960,159.3373,3.4481,0.0000
C00964=1.312,-50.962,81.916,158.0920,-0.6690,0.0000
C00965=0.000,-50.970,81.946,158.1022,-0.0005,0.0000
C00966=0.000,-50.970,81.946,158.1022,-0.0005,0.0000
C00967=-1.311,-50.962,81.916,158.0920,0.6694,0.0000
C00968=-3.454,-50.970,81.960,159.3382,-3.4501,0.0000
C00969=-6.389,-52.261,82.960,173.6413,-7.6042,0.0000
C00970=-7.633,-56.525,85.423,-179.7440,1.7649,0.0000
C00971=-8.475,-63.374,88.663,-179.7387,1.9278,0.0000
C00972=-9.515,-71.858,91.777,-179.8100,1.4311,0.0000
C00973=-10.634,-80.658,94.007,-179.8912,0.8247,0.0000
C00974=-11.808,-88.386,95.061,-179.8809,0.3884,0.0000
C00975=-15.455,-93.966,95.604,-179.9140,0.0739,0.0000
C00976=-55.516,-77.372,95.604,-179.9914,-0.1131,0.0000
C00977=-54.149,-70.847,95.061,179.8096,-0.3589,0.0000
C00978=-49.515,-64.553,94.007,179.4937,-0.6602,0.0000
C00979=-44.083,-57.539,91.777,179.1223,-1.1463,0.0000
C00980=-38.820,-50.805,88.663,178.8213,-1.5481,0.0000
C00981=-34.571,-45.367,85.423,178.9328,-1.4291,0.0000
C00982=-32.436,-41.472,82.960,-179.1064,9.8268,0.0000
C00983=-33.599,-38.483,81.960,167.3708,17.1854,0.0000
C00984=-35.108,-36.963,81.916,163.6891,15.4355,0.0000
C00985=-36.041,-36.041,81.946,164.1333,15.8661,0.0000
C00986=-36.963,-35.108,81.916,164.5648,16.3112,0.0000
C00987=-38.483,-33.599,81.960,162.8140,12.6271,0.0000
C00988=-41.472,-32.436,82.960,170.1739,-0.8939,0.0000
C00989=-45.367,-34.571,85.423,-178.5709,1.0672,0.0000
C00990=-50.805,-38.820,88.663,-178.4519,1.1787,0.0000
C00991=-57.539,-44.083,91.777,-178.8537,0.8777,0.0000
C00992=-64.553,-49.515,94.007,-179.3398,0.5063,0.0000
C00993=-70.847,-54.149,95.061,-179.6411,0.1904,0.0000
C00994=-77.372,-55.516,95.604,-179.8869,-0.0086,0.0000
C00995=-93.966,-15.455,95.604,179.9261,-0.0860,0.0000
C00996=-88.386,-11.808,95.061,179.6116,-0.1191,0.0000
C00997=-80.658,-10.634,94.007,179.1753,-0.1088,0.0000
C00998=-71.858,-9.515,91.777,178.5689,-0.1900,0.0000
C00999=-63.374,-8.475,88.663,178.0722,-0.2613,0.0000
C01000=-56.525,-7.633,85.423,178.2351,-0.2560,0.0000
C01001=-52.261,-6.389,82.960,-172.3955,6.3594,0.0000
C01002=-50.970,-3.453,81.960,-176.5519,20.6627,0.0000
C01003=-50.962,-1.312,81.916,179.3310,21.9080,0.0000
C01004=-50.970,0.000,81.946,179.9995,21.8978,0.0000
C01005=-50.962,1.311,81.916,-179.3306,21.9080,0.0000
C01006=-50.970,3.454,81.960,176.5499,20.6618,0.0000
C01007=-52.261,6.389,82.960,172.3958,6.3587,0.0000
C01008=-56.525,7.633,85.423,-178.2351,-0.2560,0.0000
C01009=-63.374,8.475,88.663,-178.0722,-0.2613,0.0000
C01010=-71.858,9.515,91.777,-178.5689,-0.1900,0.0000
C01011=-80.658,10.634,94.007,-179.1753,-0.1088,0.0000
C01012=-88.386,11.808,95.061,-179.6116,-0.1191,0.0000
C01013=-93.966,15.455,95.604,-179.9261,-0.0860,0.0000
C01014=-77.372,55.516,95.604,179.8869,-0.0086,0.0000
C01015=-70.847,54.149,95.061,179.6411,0.1904,0.0000
C01016=-64.553,49.515,94.007,179.3398,0.5063,0.0000
C01017=-57.539,44.083,91.777,178.8537,0.8777,0.0000
C01018=-50.805,38.820,88.663,178.4519,1.1787,0.0000
C01019=-45.367,34.571,85.423,178.5709,1.0672,0.0000
C01020=-41.472,32.436,82.960,-170.1732,-0.8936,0.0000
C01021=-38.483,33.599,81.960,-162.8146,12.6292,0.0000
C01022=-36.963,35.108,81.916,-164.5645,16.3109,0.0000
C01023=-36.041,36.041,81.946,-164.1339,15.8667,0.0000
C01024=-35.108,36.963,81.916,-163.6888,15.4352,0.0000
C01025=-33.599,38.483,81.960,-167.3729,17.1860,0.0000
C01026=-32.436,41.472,82.960,179.1061,9.8261,0.0000
C01027=-34.571,45.367,85.423,-178.9328,-1.4291,0.0000
C01028=-38.820,50.805,88.663,-178.8213,-1.5481,0.0000
C01029=-44.083,57.539,91.777,-179.1223,-1.1463,0.0000
C01030=-49.515,64.553,94.007,-179.4937,-0.6602,0.0000
C01031=-54.149,70.847,95.061,-179.8096,-0.3589,0.0000
C01032=-55.516,77.372,95.604,179.9914,-0.1131,0.0000
C01033=-15.455,93.966,95.604,179.9140,0.0739,0.0000
C01034=-11.808,88.386,95.061,179.8809,0.3884,0.0000
C01035=-10.634,80.658,94.007,179.8912,0.8247,0.0000
C01036=-9.515,71.858,91.777,179.8100,1.4311,0.0000
C01037=-8.475,63.374,88.663,179.7387,1.9278,0.0000
C01038=-7.633,56.525,85.423,179.7440,1.7649,0.0000
C01039=-6.389,52.261,82.960,-173.6413,-7.6042,0.0000
C01040=-3.454,50.970,81.960,-159.3382,-3.4501,0.0000
C01041=-1.311,50.962,81.916,-158.0920,0.6694,0.0000
C01042=0.000,50.970,81.946,-158.1022,-0.0005,0.0000
C01043=0.000,50.195,84.004,-160.6619,-0.0004,0.0000
C01044=1.241,50.188,83.974,-160.6464,-0.5462,0.0000
C01045=3.334,50.204,84.019,-161.8405,3.1426,0.0000
C01046=6.253,51.571,85.045,-174.7212,6.4678,0.0000
C01047=7.499,56.017,87.559,179.7895,-1.5010,0.0000
C01048=8.371,63.087,90.842,179.8130,-1.3996,0.0000
C01049=9.459,71.748,93.974,179.9071,-0.7043,0.0000
C01050=44.045,57.421,93.974,-179.5677,0.5637,0.0000
C01051=38.690,50.529,90.842,-179.1424,1.1219,0.0000
C01052=34.307,44.912,87.559,-179.0873,1.2103,0.0000
C01053=32.045,40.888,85.045,179.1504,-8.2781,0.0000
C01054=33.142,37.857,84.019,-169.0703,-15.1499,0.0000
C01055=34.611,36.365,83.974,-165.6885,-13.5839,0.0000
C01056=35.493,35.493,84.004,-166.0631,-13.9364,0.0000
C01057=36.365,34.611,83.974,-166.4163,-14.3116,0.0000
C01058=37.858,33.142,84.019,-164.8496,-10.9278,0.0000
C01059=40.888,32.045,85.045,-171.7226,0.8499,0.0000
C01060=44.912,34.307,87.559,178.7897,-0.9127,0.0000
C01061=50.529,38.690,90.842,178.8781,-0.8576,0.0000
C01062=57.421,44.045,93.974,179.4363,-0.4323,0.0000
C01063=71.748,9.459,93.974,-179.2957,0.0929,0.0000
C01064=63.087,8.371,90.842,-178.6004,0.1870,0.0000
C01065=56.017,7.499,87.559,-178.4990,0.2105,0.0000
C01066=51.571,6.253,85.045,173.5322,-5.2788,0.0000
C01067=50.204,3.334,84.019,176.8574,-18.1595,0.0000
C01068=50.188,1.241,83.974,-179.4538,-19.3536,0.0000
C01069=50.195,0.000,84.004,-179.9996,-19.3381,0.0000
C01070=50.188,-1.240,83.974,179.4535,-19.3536,0.0000
C01071=50.204,-3.335,84.019,-176.8556,-18.1586,0.0000
C01072=51.571,-6.253,85.045,-173.5325,-5.2781,0.0000
C01073=56.017,-7.499,87.559,178.4990,0.2105,0.0000
C01074=63.087,-8.371,90.842,178.6004,0.1870,0.0000
C01075=71.748,-9.459,93.974,179.2957,0.0929,0.0000
C01076=57.421,-44.045,93.974,-179.4363,-0.4323,0.0000
C01077=50.529,-38.690,90.842,-178.8781,-0.8576,0.0000
C01078=44.912,-34.307,87.559,-178.7897,-0.9127,0.0000
C01079=40.888,-32.045,85.045,171.7219,0.8496,0.0000
C01080=37.857,-33.142,84.019,164.8501,-10.9297,0.0000
C01081=36.365,-34.611,83.974,166.4161,-14.3115,0.0000
C01082=35.493,-35.493,84.004,166.0636,-13.9369,0.0000
C01083=34.611,-36.365,83.974,165.6884,-13.5837,0.0000
C01084=33.142,-37.858,84.019,169.0722,-15.1504,0.0000
C01085=32.045,-40.888,85.045,-179.1501,-8.2774,0.0000
C01086=34.307,-44.912,87.559,179.0873,1.2103,0.0000
C01087=38.690,-50.529,90.842,179.1424,1.1219,0.0000
C01088=44.045,-57.421,93.974,179.5677,0.5637,0.0000
C01089=9.459,-71.748,93.974,-179.9071,-0.7043,0.0000
C01090=8.371,-63.087,90.842,-179.8130,-1.3996,0.0000
C01091=7.499,-56.017,87.559,-179.7895,-1.5010,0.0000
C01092=6.253,-51.571,85.045,174.7212,6.4678,0.0000
C01093=3.334,-50.204,84.019,161.8405,3.1426,0.0000
C01094=1.241,-50.188,83.974,160.6464,-0.5462,0.0000
C01095=0.000,-50.195,84.004,160.6619,-0.0004,0.0000
C01096=0.000,-50.195,84.004,160.6619,-0.0004,0.0000
C01097=-1.240,-50.188,83.974,160.6464,0.5465,0.0000
C01098=-3.335,-50.204,84.019,161.8414,-3.1444,0.0000
C01099=-6.253,-51.571,85.045,174.7219,-6.4675,0.0000
C01100=-7.499,-56.017,87.559,-179.7895,1.5010,0.0000
C01101=-8.371,-63.087,90.842,-179.8130,1.3996,0.0000
C01102=-9.459,-71.748,93.974,-179.9071,0.7043,0.0000
C01103=-44.045,-57.421,93.974,179.5677,-0.5637,0.0000
C01104=-38.690,-50.529,90.842,179.1424,-1.1219,0.0000
C01105=-34.307,-44.912,87.559,179.0873,-1.2103,0.0000
C01106=-32.045,-40.888,85.045,-179.1504,8.2781,0.0000
C01107=-33.142,-37.857,84.019,169.0703,15.1499,0.0000
C01108=-34.611,-36.365,83.974,165.6885,13.5839,0.0000
C01109=-35.493,-35.493,84.004,166.0631,13.9364,0.0000
C01110=-36.365,-34.611,83.974,166.4163,14.3116,0.0000
C01111=-37.858,-33.142,84.019,164.8496,10.9278,0.0000
C01112=-40.888,-32.045,85.045,171.7226,-0.8499,0.0000
C01113=-44.912,-34.307,87.559,-178.7897,0.9127,0.0000
C01114=-50.529,-38.690,90.842,-178.8781,0.8576,0.0000
C01115=-57.421,-44.045,93.974,-179.4363,0.4323,0.0000
C01116=-71.748,-9.459,93.974,179.2957,-0.0929,0.0000
C01117=-63.087,-8.371,90.842,178.6004,-0.1870,0.0000
C01118=-56.017,-7.499,87.559,178.4990,-0.2105,0.0000
C01119=-51.571,-6.253,85.045,-173.5322,5.2788,0.0000
C01120=-50.204,-3.334,84.019,-176.8574,18.1595,0.0000
C01121=-50.188,-1.241,83.974,179.4538,19.3536,0.0000
C01122=-50.195,0.000,84.004,179.9996,19.3381,0.0000
C01123=-50.188,1.240,83.974,-179.4535,19.3536,0.0000
C01124=-50.204,3.335,84.019,176.8556,18.1586,0.0000
C01125=-51.571,6.253,85.045,173.5325,5.2781,0.0000
C01126=-56.017,7.499,87.559,-178.4990,-0.2105,0.0000
C01127=-63.087,8.371,90.842,-178.6004,-0.1870,0.0000
C01128=-71.748,9.459,93.974,-179.2957,-0.0929,0.0000
C01129=-57.421,44.045,93.974,179.4363,0.4323,0.0000
C01130=-50.529,38.690,90.842,178.8781,0.8576,0.0000
C01131=-44.912,34.307,87.559,178.7897,0.9127,0.0000
C01132=-40.888,32.045,85.045,-171.7219,-0.8496,0.0000
C01133=-37.857,33.142,84.019,-164.8501,10.9297,0.0000
C01134=-36.365,34.611,83.974,-166.4161,14.3115,0.0000
C01135=-35.493,35.493,84.004,-166.0636,13.9369,0.0000
C01136=-34.611,36.365,83.974,-165.6884,13.5837,0.0000
C01137=-33.142,37.858,84.019,-169.0722,15.1504,0.0000
C01138=-32.045,40.888,85.045,179.1501,8.2774,0.0000
C01139=-34.307,44.912,87.559,-179.0873,-1.2103,0.0000
C01140=-38.690,50.529,90.842,-179.1424,-1.1219,0.0000
C01141=-44.045,57.421,93.974,-179.5677,-0.5637,0.0000
C01142=-9.459,71.748,93.974,179.9071,0.7043,0.0000
C01143=-8.371,63.087,90.842,179.8130,1.3996,0.0000
C01144=-7.499,56.017,87.559,179.7895,1.5010,0.0000
C01145=-6.253,51.571,85.045,-174.7219,-6.4675,0.0000
C01146=-3.335,50.204,84.019,-161.8414,-3.1444,0.0000
C01147=-1.240,50.188,83.974,-160.6464,0.5465,0.0000
C01148=0.000,50.195,84.004,-160.6619,-0.0004,0.0000
C01149=0.000,49.517,86.097,-163.4981,-0.0002,0.0000
C01150=1.179,49.510,86.067,-163.4764,-0.4305,0.0000
C01151=3.230,49.536,86.112,-164.5770,2.7513,0.0000
C01152=6.137,50.981,87.161,-175.7739,5.2863,0.0000
C01153=7.391,55.610,89.719,179.8393,-1.1782,0.0000
C01154=8.302,62.896,93.033,179.8904,-0.8284,0.0000
C01155=38.603,50.345,93.033,-179.4917,0.6633,0.0000
C01156=34.096,44.548,89.719,-179.2805,0.9468,0.0000
C01157=31.710,40.389,87.161,179.2451,-6.7115,0.0000
C01158=32.743,37.311,86.112,-170.8486,-12.9014,0.0000
C01159=34.176,35.843,86.067,-167.8615,-11.5554,0.0000
C01160=35.014,35.014,86.097,-168.1686,-11.8311,0.0000
C01161=35.842,34.176,86.067,-168.4447,-12.1386,0.0000
C01162=37.311,32.743,86.112,-167.0982,-9.1497,0.0000
C01163=40.389,31.710,87.161,-173.2891,0.7551,0.0000
C01164=44.548,34.096,89.719,179.0532,-0.7195,0.0000
C01165=50.345,38.603,93.033,179.3367,-0.5083,0.0000
C01166=62.896,8.302,93.033,-179.1716,0.1096,0.0000
C01167=55.610,7.391,89.719,-178.8218,0.1607,0.0000
C01168=50.981,6.137,87.161,174.7137,-4.2261,0.0000
C01169=49.536,3.230,86.112,177.2487,-15.4230,0.0000
C01170=49.510,1.179,86.067,-179.5695,-16.5236,0.0000
C01171=49.517,0.000,86.097,-179.9998,-16.5019,0.0000
C01172=49.510,-1.178,86.067,179.5694,-16.5236,0.0000
C01173=49.536,-3.231,86.112,-177.2471,-15.4221,0.0000
C01174=50.981,-6.137,87.161,-174.7140,-4.2255,0.0000
C01175=55.610,-7.391,89.719,178.8218,0.1607,0.0000
C01176=62.896,-8.302,93.033,179.1716,0.1096,0.0000
C01177=50.345,-38.603,93.033,-179.3367,-0.5083,0.0000
C01178=44.548,-34.096,89.719,-179.0532,-0.7195,0.0000
C01179=40.389,-31.710,87.161,173.2885,0.7549,0.0000
C01180=37.311,-32.743,86.112,167.0986,-9.1514,0.0000
C01181=35.843,-34.176,86.067,168.4446,-12.1385,0.0000
C01182=35.014,-35.014,86.097,168.1689,-11.8314,0.0000
C01183=34.176,-35.842,86.067,167.8614,-11.5553,0.0000
C01184=32.743,-37.311,86.112,170.8503,-12.9018,0.0000
C01185=31.710,-40.389,87.161,-179.2449,-6.7109,0.0000
C01186=34.096,-44.548,89.719,179.2805,0.9468,0.0000
C01187=38.603,-50.345,93.033,179.4917,0.6633,0.0000
C01188=8.302,-62.896,93.033,-179.8904,-0.8284,0.0000
C01189=7.391,-55.610,89.719,-179.8393,-1.1782,0.0000
C01190=6.137,-50.981,87.161,175.7739,5.2863,0.0000
C01191=3.230,-49.536,86.112,164.5770,2.7513,0.0000
C01192=1.179,-49.510,86.067,163.4764,-0.4305,0.0000
C01193=0.000,-49.517,86.097,163.4981,-0.0002,0.0000
C01194=0.000,-49.517,86.097,163.4981,-0.0002,0.0000
C01195=-1.178,-49.510,86.067,163.4764,0.4306,0.0000
C01196=-3.231,-49.536,86.112,164.5779,-2.7529,0.0000
C01197=-6.137,-50.981,87.161,175.7745,-5.2860,0.0000
C01198=-7.391,-55.610,89.719,-179.8393,1.1782,0.0000
C01199=-8.302,-62.896,93.033,-179.8904,0.8284,0.0000
C01200=-38.603,-50.345,93.033,179.4917,-0.6633,0.0000
C01201=-34.096,-44.548,89.719,179.2805,-0.9468,0.0000
C01202=-31.710,-40.389,87.161,-179.2451,6.7115,0.0000
C01203=-32.743,-37.311,86.112,170.8486,12.9014,0.0000
C01204=-34.176,-35.843,86.067,167.8615,11.5554,0.0000
C01205=-35.014,-35.014,86.097,168.1686,11.8311,0.0000
C01206=-35.842,-34.176,86.067,168.4447,12.1386,0.0000
C01207=-37.311,-32.743,86.112,167.0982,9.1497,0.0000
C01208=-40.389,-31.710,87.161,173.2891,-0.7551,0.0000
C01209=-44.548,-34.096,89.719,-179.0532,0.7195,0.0000
C01210=-50.345,-38.603,93.033,-179.3367,0.5083,0.0000
C01211=-62.896,-8.302,93.033,179.1716,-0.1096,0.0000
C01212=-55.610,-7.391,89.719,178.8218,-0.1607,0.0000
C01213=-50.981,-6.137,87.161,-174.7137,4.2261,0.0000
C01214=-49.536,-3.230,86.112,-177.2487,15.4230,0.0000
C01215=-49.510,-1.179,86.067,179.5695,16.5236,0.0000
C01216=-49.517,0.000,86.097,179.9998,16.5019,0.0000
C01217=-49.510,1.178,86.067,-179.5694,16.5236,0.0000
C01218=-49.536,3.231,86.112,177.2471,15.4221,0.0000
C01219=-50.981,6.137,87.161,174.7140,4.2255,0.0000
C01220=-55.610,7.391,89.719,-178.8218,-0.1607,0.0000
C01221=-62.896,8.302,93.033,-179.1716,-0.1096,0.0000
C01222=-50.345,38.603,93.033,179.3367,0.5083,0.0000
C01223=-44.548,34.096,89.719,179.0532,0.7195,0.0000
C01224=-40.389,31.710,87.161,-173.2885,-0.7549,0.0000
C01225=-37.311,32.743,86.112,-167.0986,9.1514,0.0000
C01226=-35.843,34.176,86.067,-168.4446,12.1385,0.0000
C01227=-35.014,35.014,86.097,-168.1689,11.8314,0.0000
C01228=-34.176,35.842,86.067,-167.8614,11.5553,0.0000
C01229=-32.743,37.311,86.112,-170.8503,12.9018,0.0000
C01230=-31.710,40.389,87.161,179.2449,6.7109,0.0000
C01231=-34.096,44.548,89.719,-179.2805,-0.9468,0.0000
C01232=-38.603,50.345,93.033,-179.4917,-0.6633,0.0000
C01233=-8.302,62.896,93.033,179.8904,0.8284,0.0000
C01234=-7.391,55.610,89.719,179.8393,1.1782,0.0000
C01235=-6.137,50.981,87.161,-175.7745,-5.2860,0.0000
C01236=-3.231,49.536,86.112,-164.5779,-2.7529,0.0000
C01237=-1.178,49.510,86.067,-163.4764,0.4306,0.0000
C01238=0.000,49.517,86.097,-163.4981,-0.0002,0.0000
C01239=0.000,48.949,88.223,-166.6221,-0.0001,0.0000
C01240=1.127,48.942,88.191,-166.5931,-0.3233,0.0000
C01241=3.143,48.975,88.238,-167.5529,2.2752,0.0000
C01242=6.042,50.501,89.306,-176.8083,4.0597,0.0000
C01243=7.312,55.314,91.898,179.8925,-0.8037,0.0000
C01244=8.270,62.805,95.231,179.9710,-0.2201,0.0000
C01245=38.562,50.258,95.231,-179.8648,0.1762,0.0000
C01246=33.942,44.284,91.898,-179.5076,0.6443,0.0000
C01247=31.437,39.982,89.306,179.3837,-5.1210,0.0000
C01248=32.408,36.853,88.238,-172.7068,-10.4353,0.0000
C01249=33.811,35.404,88.191,-170.2108,-9.3446,0.0000
C01250=34.612,34.612,88.223,-170.4539,-9.5459,0.0000
C01251=35.404,33.811,88.191,-170.6554,-9.7892,0.0000
C01252=36.854,32.408,88.238,-169.5644,-7.2918,0.0000
C01253=39.982,31.437,89.306,-174.8795,0.6164,0.0000
C01254=44.284,33.942,91.898,179.3557,-0.4924,0.0000
C01255=50.258,38.562,95.231,179.8238,-0.1352,0.0000
C01256=62.805,8.270,95.231,-179.7799,0.0290,0.0000
C01257=55.314,7.312,91.898,-179.1963,0.1075,0.0000
C01258=50.501,6.042,89.306,175.9403,-3.1917,0.0000
C01259=48.975,3.143,88.238,177.7248,-12.4471,0.0000
C01260=48.942,1.127,88.191,-179.6767,-13.4069,0.0000
C01261=48.949,0.000,88.223,-179.9999,-13.3779,0.0000
C01262=48.942,-1.126,88.191,179.6767,-13.4069,0.0000
C01263=48.976,-3.143,88.238,-177.7235,-12.4463,0.0000
C01264=50.501,-6.042,89.306,-175.9405,-3.1912,0.0000
C01265=55.314,-7.312,91.898,179.1963,0.1075,0.0000
C01266=62.805,-8.270,95.231,179.7799,0.0290,0.0000
C01267=50.258,-38.562,95.231,-179.8238,-0.1352,0.0000
C01268=44.284,-33.942,91.898,-179.3557,-0.4924,0.0000
C01269=39.982,-31.437,89.306,174.8790,0.6163,0.0000
C01270=36.853,-32.408,88.238,169.5647,-7.2932,0.0000
C01271=35.404,-33.811,88.191,170.6554,-9.7892,0.0000
C01272=34.612,-34.612,88.223,170.4541,-9.5461,0.0000
C01273=33.811,-35.404,88.191,170.2108,-9.3446,0.0000
C01274=32.408,-36.854,88.238,172.7082,-10.4356,0.0000
C01275=31.437,-39.982,89.306,-179.3836,-5.1205,0.0000
C01276=33.942,-44.284,91.898,179.5076,0.6443,0.0000
C01277=38.562,-50.258,95.231,179.8648,0.1762,0.0000
C01278=8.270,-62.805,95.231,-179.9710,-0.2201,0.0000
C01279=7.312,-55.314,91.898,-179.8925,-0.8037,0.0000
C01280=6.042,-50.501,89.306,176.8083,4.0597,0.0000
C01281=3.143,-48.975,88.238,167.5529,2.2752,0.0000
C01282=1.127,-48.942,88.191,166.5931,-0.3233,0.0000
C01283=0.000,-48.949,88.223,166.6221,-0.0001,0.0000
C01284=0.000,-48.949,88.223,166.6221,-0.0001,0.0000
C01285=-1.126,-48.942,88.191,166.5931,0.3233,0.0000
C01286=-3.143,-48.976,88.238,167.5537,-2.2765,0.0000
C01287=-6.042,-50.501,89.306,176.8088,-4.0595,0.0000
C01288=-7.312,-55.314,91.898,-179.8925,0.8037,0.0000
C01289=-8.270,-62.805,95.231,-179.9710,0.2201,0.0000
C01290=-38.562,-50.258,95.231,179.8648,-0.1762,0.0000
C01291=-33.942,-44.284,91.898,179.5076,-0.6443,0.0000
C01292=-31.437,-39.982,89.306,-179.3837,5.1210,0.0000
C01293=-32.408,-36.853,88.238,172.7068,10.4353,0.0000
C01294=-33.811,-35.404,88.191,170.2108,9.3446,0.0000
C01295=-34.612,-34.612,88.223,170.4539,9.5459,0.0000
C01296=-35.404,-33.811,88.191,170.6554,9.7892,0.0000
C01297=-36.854,-32.408,88.238,169.5644,7.2918,0.0000
C01298=-39.982,-31.437,89.306,174.8795,-0.6164,0.0000
C01299=-44.284,-33.942,91.898,-179.3557,0.4924,0.0000
C01300=-50.258,-38.562,95.231,-179.8238,0.1352,0.0000
C01301=-62.805,-8.270,95.231,179.7799,-0.0290,0.0000
C01302=-55.314,-7.312,91.898,179.1963,-0.1075,0.0000
C01303=-50.501,-6.042,89.306,-175.9403,3.1917,0.0000
C01304=-48.975,-3.143,88.238,-177.7248,12.4471,0.0000
C01305=-48.942,-1.127,88.191,179.6767,13.4069,0.0000
C01306=-48.949,0.000,88.223,179.9999,13.3779,0.0000
C01307=-48.942,1.126,88.191,-179.6767,13.4069,0.0000
C01308=-48.976,3.143,88.238,177.7235,12.4463,0.0000
C01309=-50.501,6.042,89.306,175.9405,3.1912,0.0000
C01310=-55.314,7.312,91.898,-179.1963,-0.1075,0.0000
C01311=-62.805,8.270,95.231,-179.7799,-0.0290,0.0000
C01312=-50.258,38.562,95.231,179.8238,0.1352,0.0000
C01313=-44.284,33.942,91.898,179.3557,0.4924,0.0000
C01314=-39.982,31.437,89.306,-174.8790,-0.6163,0.0000
C01315=-36.853,32.408,88.238,-169.5647,7.2932,0.0000
C01316=-35.404,33.811,88.191,-170.6554,9.7892,0.0000
C01317=-34.612,34.612,88.223,-170.4541,9.5461,0.0000
C01318=-33.811,35.404,88.191,-170.2108,9.3446,0.0000
C01319=-32.408,36.854,88.238,-172.7082,10.4356,0.0000
C01320=-31.437,39.982,89.306,179.3836,5.1205,0.0000
C01321=-33.942,44.284,91.898,-179.5076,-0.6443,0.0000
C01322=-38.562,50.258,95.231,-179.8648,-0.1762,0.0000
C01323=-8.270,62.805,95.231,179.9710,0.2201,0.0000
C01324=-7.312,55.314,91.898,179.8925,0.8037,0.0000
C01325=-6.042,50.501,89.306,-176.8088,-4.0595,0.0000
C01326=-3.143,48.976,88.238,-167.5537,-2.2765,0.0000
C01327=-1.126,48.942,88.191,-166.5931,0.3233,0.0000
C01328=0.000,48.949,88.223,-166.6221,-0.0001,0.0000
C01329=0.000,48.503,90.377,-170.0356,-0.0001,0.0000
C01330=1.086,48.496,90.345,-169.9984,-0.2252,0.0000
C01331=3.075,48.536,90.393,-170.7679,1.7188,0.0000
C01332=5.972,50.143,91.476,-177.8365,2.7864,0.0000
C01333=7.266,55.138,94.090,179.9489,-0.3871,0.0000
C01334=33.851,44.126,94.090,-179.7624,0.3099,0.0000
C01335=31.234,39.679,91.476,179.5587,-3.4981,0.0000
C01336=32.146,36.494,90.393,-174.6463,-7.7532,0.0000
C01337=33.524,35.059,90.345,-172.7350,-6.9514,0.0000
C01338=34.297,34.297,90.377,-172.9184,-7.0815,0.0000
C01339=35.059,33.525,90.345,-173.0486,-7.2649,0.0000
C01340=36.495,32.146,90.393,-172.2466,-5.3526,0.0000
C01341=39.679,31.234,91.476,-176.5023,0.4414,0.0000
C01342=44.126,33.851,94.090,179.6901,-0.2376,0.0000
C01343=55.138,7.266,94.090,-179.6129,0.0511,0.0000
C01344=50.143,5.972,91.476,177.2136,-2.1635,0.0000
C01345=48.536,3.075,90.393,178.2812,-9.2321,0.0000
C01346=48.496,1.086,90.345,-179.7748,-10.0016,0.0000
C01347=48.503,0.000,90.377,-179.9999,-9.9644,0.0000
C01348=48.496,-1.085,90.345,179.7749,-10.0016,0.0000
C01349=48.536,-3.075,90.393,-178.2802,-9.2314,0.0000
C01350=50.143,-5.972,91.476,-177.2137,-2.1632,0.0000
C01351=55.138,-7.266,94.090,179.6129,0.0511,0.0000
C01352=44.126,-33.851,94.090,-179.6901,-0.2376,0.0000
C01353=39.679,-31.234,91.476,176.5019,0.4413,0.0000
C01354=36.494,-32.146,90.393,172.2468,-5.3537,0.0000
C01355=35.059,-33.524,90.345,173.0486,-7.2650,0.0000
C01356=34.297,-34.297,90.377,172.9185,-7.0816,0.0000
C01357=33.525,-35.059,90.345,172.7351,-6.9514,0.0000
C01358=32.146,-36.495,90.393,174.6474,-7.7534,0.0000
C01359=31.234,-39.679,91.476,-179.5586,-3.4977,0.0000
C01360=33.851,-44.126,94.090,179.7624,0.3099,0.0000
C01361=7.266,-55.138,94.090,-179.9489,-0.3871,0.0000
C01362=5.972,-50.143,91.476,177.8365,2.7864,0.0000
C01363=3.075,-48.536,90.393,170.7679,1.7188,0.0000
C01364=1.086,-48.496,90.345,169.9984,-0.2252,0.0000
C01365=0.000,-48.503,90.377,170.0356,-0.0001,0.0000
C01366=0.000,-48.503,90.377,170.0356,-0.0001,0.0000
C01367=-1.085,-48.496,90.345,169.9984,0.2251,0.0000
C01368=-3.075,-48.536,90.393,170.7686,-1.7198,0.0000
C01369=-5.972,-50.143,91.476,177.8368,-2.7863,0.0000
C01370=-7.266,-55.138,94.090,-179.9489,0.3871,0.0000
C01371=-33.851,-44.126,94.090,179.7624,-0.3099,0.0000
C01372=-31.234,-39.679,91.476,-179.5587,3.4981,0.0000
C01373=-32.146,-36.494,90.393,174.6463,7.7532,0.0000
C01374=-33.524,-35.059,90.345,172.7350,6.9514,0.0000
C01375=-34.297,-34.297,90.377,172.9184,7.0815,0.0000
C01376=-35.059,-33.525,90.345,173.0486,7.2649,0.0000
C01377=-36.495,-32.146,90.393,172.2466,5.3526,0.0000
C01378=-39.679,-31.234,91.476,176.5023,-0.4414,0.0000
C01379=-44.126,-33.851,94.090,-179.6901,0.2376,0.0000
C01380=-55.138,-7.266,94.090,179.6129,-0.0511,0.0000
C01381=-50.143,-5.972,91.476,-177.2136,2.1635,0.0000
C01382=-48.536,-3.075,90.393,-178.2812,9.2321,0.0000
C01383=-48.496,-1.086,90.345,179.7748,10.0016,0.0000
C01384=-48.503,0.000,90.377,179.9999,9.9644,0.0000
C01385=-48.496,1.085,90.345,-179.7749,10.0016,0.0000
C01386=-48.536,3.075,90.393,178.2802,9.2314,0.0000
C01387=-50.143,5.972,91.476,177.2137,2.1632,0.0000
C01388=-55.138,7.266,94.090,-179.6129,-0.0511,0.0000
C01389=-44.126,33.851,94.090,179.6901,0.2376,0.0000
C01390=-39.679,31.234,91.476,-176.5019,-0.4413,0.0000
C01391=-36.494,32.146,90.393,-172.2468,5.3537,0.0000
C01392=-35.059,33.524,90.345,-173.0486,7.2650,0.0000
C01393=-34.297,34.297,90.377,-172.9185,7.0816,0.0000
C01394=-33.525,35.059,90.345,-172.7351,6.9514,0.0000
C01395=-32.146,36.495,90.393,-174.6474,7.7534,0.0000
C01396=-31.234,39.679,91.476,179.5586,3.4977,0.0000
C01397=-33.851,44.126,94.090,-179.7624,-0.3099,0.0000
C01398=-7.266,55.138,94.090,179.9489,0.3871,0.0000
C01399=-5.972,50.143,91.476,-177.8368,-2.7863,0.0000
C01400=-3.075,48.536,90.393,-170.7686,-1.7198,0.0000
C01401=-1.085,48.496,90.345,-169.9984,0.2251,0.0000
C01402=0.000,48.503,90.377,-170.0356,-0.0001,0.0000
C01403=0.000,48.191,92.555,-173.7266,-0.0000,0.0000
C01404=1.057,48.183,92.523,-173.6804,-0.1349,0.0000
C01405=3.027,48.229,92.571,-174.2129,1.0909,0.0000
C01406=5.927,49.917,93.664,-178.8724,1.4637,0.0000
C01407=31.106,39.488,93.664,179.7623,-1.8320,0.0000
C01408=31.963,36.244,92.571,-176.6691,-4.8658,0.0000
C01409=33.323,34.818,92.523,-175.4275,-4.3829,0.0000
C01410=34.076,34.076,92.555,-175.5552,-4.4448,0.0000
C01411=34.818,33.324,92.523,-175.6171,-4.5724,0.0000
C01412=36.244,31.963,92.571,-175.1341,-3.3301,0.0000
C01413=39.488,31.106,93.664,-178.1682,0.2378,0.0000
C01414=49.917,5.927,93.664,178.5363,-1.1276,0.0000
C01415=48.229,3.027,92.571,178.9091,-5.7871,0.0000
C01416=48.183,1.057,92.523,-179.8651,-6.3196,0.0000
C01417=48.191,0.000,92.555,-180.0000,-6.2734,0.0000
C01418=48.183,-1.057,92.523,179.8652,-6.3196,0.0000
C01419=48.229,-3.027,92.571,-178.9086,-5.7866,0.0000
C01420=49.918,-5.927,93.664,-178.5365,-1.1274,0.0000
C01421=39.488,-31.106,93.664,178.1680,0.2377,0.0000
C01422=36.244,-31.963,92.571,175.1342,-3.3309,0.0000
C01423=34.818,-33.323,92.523,175.6171,-4.5725,0.0000
C01424=34.076,-34.076,92.555,175.5552,-4.4448,0.0000
C01425=33.324,-34.818,92.523,175.4276,-4.3829,0.0000
C01426=31.963,-36.244,92.571,176.6699,-4.8659,0.0000
C01427=31.106,-39.488,93.664,-179.7622,-1.8318,0.0000
C01428=5.927,-49.917,93.664,178.8724,1.4637,0.0000
C01429=3.027,-48.229,92.571,174.2129,1.0909,0.0000
C01430=1.057,-48.183,92.523,173.6804,-0.1349,0.0000
C01431=0.000,-48.191,92.555,173.7266,-0.0000,0.0000
C01432=0.000,-48.191,92.555,173.7266,-0.0000,0.0000
C01433=-1.057,-48.183,92.523,173.6804,0.1348,0.0000
C01434=-3.027,-48.229,92.571,174.2134,-1.0914,0.0000
C01435=-5.927,-49.918,93.664,178.8726,-1.4635,0.0000
C01436=-31.106,-39.488,93.664,-179.7623,1.8320,0.0000
C01437=-31.963,-36.244,92.571,176.6691,4.8658,0.0000
C01438=-33.323,-34.818,92.523,175.4275,4.3829,0.0000
C01439=-34.076,-34.076,92.555,175.5552,4.4448,0.0000
C01440=-34.818,-33.324,92.523,175.6171,4.5724,0.0000
C01441=-36.244,-31.963,92.571,175.1341,3.3301,0.0000
C01442=-39.488,-31.106,93.664,178.1682,-0.2378,0.0000
C01443=-49.917,-5.927,93.664,-178.5363,1.1276,0.0000
C01444=-48.229,-3.027,92.571,-178.9091,5.7871,0.0000
C01445=-48.183,-1.057,92.523,179.8651,6.3196,0.0000
C01446=-48.191,0.000,92.555,180.0000,6.2734,0.0000
C01447=-48.183,1.057,92.523,-179.8652,6.3196,0.0000
C01448=-48.229,3.027,92.571,178.9086,5.7866,0.0000
C01449=-49.918,5.927,93.664,178.5365,1.1274,0.0000
C01450=-39.488,31.106,93.664,-178.1680,-0.2377,0.0000
C01451=-36.244,31.963,92.571,-175.1342,3.3309,0.0000
C01452=-34.818,33.323,92.523,-175.6171,4.5725,0.0000
C01453=-34.076,34.076,92.555,-175.5552,4.4448,0.0000
C01454=-33.324,34.818,92.523,-175.4276,4.3829,0.0000
C01455=-31.963,36.244,92.571,-176.6699,4.8659,0.0000
C01456=-31.106,39.488,93.664,179.7622,1.8318,0.0000
C01457=-5.927,49.918,93.664,-178.8726,-1.4635,0.0000
C01458=-3.027,48.229,92.571,-174.2134,-1.0914,0.0000
C01459=-1.057,48.183,92.523,-173.6804,0.1348,0.0000
C01460=0.000,48.191,92.555,-173.7266,-0.0000,0.0000
C01461=0.000,48.026,94.749,-177.6660,-0.0000,0.0000
C01462=1.042,48.016,94.716,-177.6104,-0.0495,0.0000
C01463=3.002,48.067,94.764,-177.8674,0.4046,0.0000
C01464=5.911,49.834,95.862,-179.9324,0.0880,0.0000
C01465=31.058,39.418,95.862,179.9856,-0.1101,0.0000
C01466=31.866,36.111,94.764,-178.7776,-1.7942,0.0000
C01467=33.216,34.689,94.716,-178.2749,-1.6552,0.0000
C01468=33.959,33.959,94.749,-178.3492,-1.6508,0.0000
C01469=34.689,33.216,94.716,-178.3447,-1.7251,0.0000
C01470=36.111,31.865,94.764,-178.2059,-1.2221,0.0000
C01471=39.418,31.058,95.862,-179.8900,0.0144,0.0000
C01472=49.834,5.911,95.862,179.9120,-0.0676,0.0000
C01473=48.067,3.002,94.764,179.5954,-2.1326,0.0000
C01474=48.016,1.042,94.716,-179.9505,-2.3896,0.0000
C01475=48.026,0.000,94.749,-180.0000,-2.3340,0.0000
C01476=48.016,-1.041,94.716,179.9506,-2.3896,0.0000
C01477=48.067,-3.002,94.764,-179.5952,-2.1323,0.0000
C01478=49.834,-5.911,95.862,-179.9120,-0.0676,0.0000
C01479=39.418,-31.058,95.862,179.8899,0.0144,0.0000
C01480=36.111,-31.866,94.764,178.2058,-1.2224,0.0000
C01481=34.689,-33.216,94.716,178.3448,-1.7251,0.0000
C01482=33.959,-33.959,94.749,178.3492,-1.6508,0.0000
C01483=33.216,-34.689,94.716,178.2749,-1.6553,0.0000
C01484=31.865,-36.111,94.764,178.7779,-1.7941,0.0000
C01485=31.058,-39.418,95.862,-179.9856,-0.1100,0.0000
C01486=5.911,-49.834,95.862,179.9324,0.0880,0.0000
C01487=3.002,-48.067,94.764,177.8674,0.4046,0.0000
C01488=1.042,-48.016,94.716,177.6104,-0.0495,0.0000
C01489=0.000,-48.026,94.749,177.6660,-0.0000,0.0000
C01490=0.000,-48.026,94.749,177.6660,-0.0000,0.0000
C01491=-1.041,-48.016,94.716,177.6104,0.0494,0.0000
C01492=-3.002,-48.067,94.764,177.8677,-0.4048,0.0000
C01493=-5.911,-49.834,95.862,179.9324,-0.0880,0.0000
C01494=-31.058,-39.418,95.862,-179.9856,0.1101,0.0000
C01495=-31.866,-36.111,94.764,178.7776,1.7942,0.0000
C01496=-33.216,-34.689,94.716,178.2749,1.6552,0.0000
C01497=-33.959,-33.959,94.749,178.3492,1.6508,0.0000
C01498=-34.689,-33.216,94.716,178.3447,1.7251,0.0000
C01499=-36.111,-31.865,94.764,178.2059,1.2221,0.0000
C01500=-39.418,-31.058,95.862,179.8900,-0.0144,0.0000
C01501=-49.834,-5.911,95.862,-179.9120,0.0676,0.0000
C01502=-48.067,-3.002,94.764,-179.5954,2.1326,0.0000
C01503=-48.016,-1.042,94.716,179.9505,2.3896,0.0000
C01504=-48.026,0.000,94.749,180.0000,2.3340,0.0000
C01505=-48.016,1.041,94.716,-179.9506,2.3896,0.0000
C01506=-48.067,3.002,94.764,179.5952,2.1323,0.0000
C01507=-49.834,5.911,95.862,179.9120,0.0676,0.0000
C01508=-39.418,31.058,95.862,-179.8899,-0.0144,0.0000
C01509=-36.111,31.866,94.764,-178.2058,1.2224,0.0000
C01510=-34.689,33.216,94.716,-178.3448,1.7251,0.0000
C01511=-33.959,33.959,94.749,-178.3492,1.6508,0.0000
C01512=-33.216,34.689,94.716,-178.2749,1.6553,0.0000
C01513=-31.865,36.111,94.764,-178.7779,1.7941,0.0000
C01514=-31.058,39.418,95.862,179.9856,0.1100,0.0000
C01515=-5.911,49.834,95.862,-179.9324,-0.0880,0.0000
C01516=-3.002,48.067,94.764,-177.8677,-0.4048,0.0000
C01517=-1.041,48.016,94.716,-177.6104,0.0494,0.0000
C01518=0.000,48.026,94.749,-177.6660,-0.0000,0.0000
///TOOL 0
///POSTYPE ANGLE
///ANGLE
EC00000=-143.1205,0.0000
EC00001=-143.1463,0.0000
EC00002=-142.3113,0.0000
EC00003=-139.3171,0.0000
EC00004=-136.8101,0.0000
EC00005=-135.0000,0.0000
EC00006=-133.1899,0.0000
EC00007=-130.6822,0.0000
EC00008=-127.6881,0.0000
EC00009=-126.8537,0.0000
EC00010=-126.8795,0.0000
EC00011=-127.0066,0.0000
EC00012=-127.1043,0.0000
EC00013=-127.0265,0.0000
EC00014=-125.3500,0.0000
EC00015=-122.3913,0.0000
EC00016=-118.6599,0.0000
EC00017=-114.5839,0.0000
EC00018=-110.4161,0.0000
EC00019=-106.3398,0.0000
EC00020=-102.6088,0.0000
EC00021=-99.6504,0.0000
EC00022=-97.9733,0.0000
EC00023=-97.8955,0.0000
EC00024=-97.9932,0.0000
EC00025=-98.1209,0.0000
EC00026=-98.1459,0.0000
EC00027=-97.3110,0.0000
EC00028=-94.3168,0.0000
EC00029=-91.8104,0.0000
EC00030=-90.0000,0.0000
EC00031=-88.1906,0.0000
EC00032=-85.6822,0.0000
EC00033=-82.6890,0.0000
EC00034=-81.8541,0.0000
EC00035=-81.8791,0.0000
EC00036=-82.0068,0.0000
EC00037=-82.1045,0.0000
EC00038=-82.0267,0.0000
EC00039=-80.3496,0.0000
EC00040=-77.3912,0.0000
EC00041=-73.6602,0.0000
EC00042=-69.5839,0.0000
EC00043=-65.4161,0.0000
EC00044=-61.3401,0.0000
EC00045=-57.6087,0.0000
EC00046=-54.6500,0.0000
EC00047=-52.9735,0.0000
EC00048=-52.8957,0.0000
EC00049=-52.9934,0.0000
EC00050=-53.1205,0.0000
EC00051=-53.1463,0.0000
EC00052=-52.3113,0.0000
EC00053=-49.3171,0.0000
EC00054=-46.8101,0.0000
EC00055=-45.0000,0.0000
EC00056=-43.1899,0.0000
EC00057=-40.6822,0.0000
EC00058=-37.6881,0.0000
EC00059=-36.8537,0.0000
EC00060=-36.8795,0.0000
EC00061=-37.0066,0.0000
EC00062=-37.1043,0.0000
EC00063=-37.0265,0.0000
EC00064=-35.3500,0.0000
EC00065=-32.3913,0.0000
EC00066=-28.6599,0.0000
EC00067=-24.5839,0.0000
EC00068=-20.4161,0.0000
EC00069=-16.3398,0.0000
EC00070=-12.6088,0.0000
EC00071=-9.6504,0.0000
EC00072=-7.9733,0.0000
EC00073=-7.8955,0.0000
EC00074=-7.9932,0.0000
EC00075=-8.1209,0.0000
EC00076=-8.1459,0.0000
EC00077=-7.3110,0.0000
EC00078=-4.3178,0.0000
EC00079=-1.8094,0.0000
EC00080=0.0000,0.0000
EC00081=0.0000,0.0000
EC00082=1.7406,0.0000
EC00083=4.2255,0.0000
EC00084=7.2387,0.0000
EC00085=8.0440,0.0000
EC00086=7.9981,0.0000
EC00087=7.8709,0.0000
EC00088=7.7793,0.0000
EC00089=7.8555,0.0000
EC00090=9.5452,0.0000
EC00091=12.5282,0.0000
EC00092=16.2898,0.0000
EC00093=20.3994,0.0000
EC00094=24.6009,0.0000
EC00095=28.7101,0.0000
EC00096=32.4718,0.0000
EC00097=35.4547,0.0000
EC00098=37.1446,0.0000
EC00099=37.2208,0.0000
EC00100=37.1290,0.0000
EC00101=37.0022,0.0000
EC00102=36.9563,0.0000
EC00103=37.7605,0.0000
EC00104=40.7744,0.0000
EC00105=43.2595,0.0000
EC00106=45.0000,0.0000
EC00107=46.7398,0.0000
EC00108=49.2256,0.0000
EC00109=52.2395,0.0000
EC00110=53.0437,0.0000
EC00111=52.9978,0.0000
EC00112=52.8710,0.0000
EC00113=52.7792,0.0000
EC00114=52.8554,0.0000
EC00115=54.5453,0.0000
EC00116=57.5282,0.0000
EC00117=61.2899,0.0000
EC00118=65.3991,0.0000
EC00119=69.6006,0.0000
EC00120=73.7102,0.0000
EC00121=77.4718,0.0000
EC00122=80.4548,0.0000
EC00123=82.1445,0.0000
EC00124=82.2207,0.0000
EC00125=82.1291,0.0000
EC00126=82.0019,0.0000
EC00127=81.9560,0.0000
EC00128=82.7613,0.0000
EC00129=85.7745,0.0000
EC00130=88.2594,0.0000
EC00131=90.0000,0.0000
EC00132=91.7396,0.0000
EC00133=94.2255,0.0000
EC00134=97.2387,0.0000
EC00135=98.0440,0.0000
EC00136=97.9981,0.0000
EC00137=97.8709,0.0000
EC00138=97.7793,0.0000
EC00139=97.8555,0.0000
EC00140=99.5452,0.0000
EC00141=102.5282,0.0000
EC00142=106.2898,0.0000
EC00143=110.3994,0.0000
EC00144=114.6009,0.0000
EC00145=118.7101,0.0000
EC00146=122.4718,0.0000
EC00147=125.4547,0.0000
EC00148=127.1446,0.0000
EC00149=127.2208,0.0000
EC00150=127.1290,0.0000
EC00151=127.0022,0.0000
EC00152=126.9563,0.0000
EC00153=127.7605,0.0000
EC00154=130.7744,0.0000
EC00155=133.2595,0.0000
EC00156=135.0000,0.0000
EC00157=136.7398,0.0000
EC00158=139.2256,0.0000
EC00159=142.2395,0.0000
EC00160=143.0437,0.0000
EC00161=142.9978,0.0000
EC00162=142.8710,0.0000
EC00163=142.7792,0.0000
EC00164=142.8554,0.0000
EC00165=144.5453,0.0000
EC00166=147.5282,0.0000
EC00167=151.2899,0.0000
EC00168=155.3991,0.0000
EC00169=159.6006,0.0000
EC00170=163.7102,0.0000
EC00171=167.4718,0.0000
EC00172=170.4548,0.0000
EC00173=172.1445,0.0000
EC00174=172.2207,0.0000
EC00175=172.1291,0.0000
EC00176=172.0019,0.0000
EC00177=171.9560,0.0000
EC00178=172.7613,0.0000
EC00179=175.7745,0.0000
EC00180=178.2594,0.0000
EC00181=180.0000,0.0000
EC00182=180.0000,0.0000
EC00183=-178.2604,0.0000
EC00184=-175.7745,0.0000
EC00185=-172.7613,0.0000
EC00186=-171.9560,0.0000
EC00187=-172.0019,0.0000
EC00188=-172.1291,0.0000
EC00189=-172.2207,0.0000
EC00190=-172.1445,0.0000
EC00191=-170.4548,0.0000
EC00192=-167.4718,0.0000
EC00193=-163.7102,0.0000
EC00194=-159.6006,0.0000
EC00195=-155.3991,0.0000
EC00196=-151.2899,0.0000
EC00197=-147.5282,0.0000
EC00198=-144.5453,0.0000
EC00199=-142.8554,0.0000
EC00200=-142.7792,0.0000
EC00201=-142.8710,0.0000
EC00202=-142.9978,0.0000
EC00203=-143.0437,0.0000
EC00204=-142.2395,0.0000
EC00205=-139.2256,0.0000
EC00206=-136.7405,0.0000
EC00207=-135.0000,0.0000
EC00208=-133.2602,0.0000
EC00209=-130.7744,0.0000
EC00210=-127.7605,0.0000
EC00211=-126.9563,0.0000
EC00212=-127.0022,0.0000
EC00213=-127.1290,0.0000
EC00214=-127.2208,0.0000
EC00215=-127.1446,0.0000
EC00216=-125.4547,0.0000
EC00217=-122.4718,0.0000
EC00218=-118.7101,0.0000
EC00219=-114.6009,0.0000
EC00220=-110.3994,0.0000
EC00221=-106.2898,0.0000
EC00222=-102.5282,0.0000
EC00223=-99.5452,0.0000
EC00224=-97.8555,0.0000
EC00225=-97.7793,0.0000
EC00226=-97.8709,0.0000
EC00227=-97.9981,0.0000
EC00228=-98.0440,0.0000
EC00229=-97.2387,0.0000
EC00230=-94.2255,0.0000
EC00231=-91.7406,0.0000
EC00232=-90.0000,0.0000
EC00233=-88.2604,0.0000
EC00234=-85.7745,0.0000
EC00235=-82.7613,0.0000
EC00236=-81.9560,0.0000
EC00237=-82.0019,0.0000
EC00238=-82.1291,0.0000
EC00239=-82.2207,0.0000
EC00240=-82.1445,0.0000
EC00241=-80.4548,0.0000
EC00242=-77.4718,0.0000
EC00243=-73.7102,0.0000
EC00244=-69.6006,0.0000
EC00245=-65.3991,0.0000
EC00246=-61.2899,0.0000
EC00247=-57.5282,0.0000
EC00248=-54.5453,0.0000
EC00249=-52.8554,0.0000
EC00250=-52.7792,0.0000
EC00251=-52.8710,0.0000
EC00252=-52.9978,0.0000
EC00253=-53.0437,0.0000
EC00254=-52.2395,0.0000
EC00255=-49.2256,0.0000
EC00256=-46.7405,0.0000
EC00257=-45.0000,0.0000
EC00258=-43.2602,0.0000
EC00259=-40.7744,0.0000
EC00260=-37.7605,0.0000
EC00261=-36.9563,0.0000
EC00262=-37.0022,0.0000
EC00263=-37.1290,0.0000
EC00264=-37.2208,0.0000
EC00265=-37.1446,0.0000
EC00266=-35.4547,0.0000
EC00267=-32.4718,0.0000
EC00268=-28.7101,0.0000
EC00269=-24.6009,0.0000
EC00270=-20.3994,0.0000
EC00271=-16.2898,0.0000
EC00272=-12.5282,0.0000
EC00273=-9.5452,0.0000
EC00274=-7.8555,0.0000
EC00275=-7.7793,0.0000
EC00276=-7.8709,0.0000
EC00277=-7.9981,0.0000
EC00278=-8.0440,0.0000
EC00279=-7.2387,0.0000
EC00280=-4.2255,0.0000
EC00281=-1.7396,0.0000
EC00282=0.0000,0.0000
EC00283=0.0000,0.0000
EC00284=1.6706,0.0000
EC00285=4.1339,0.0000
EC00286=7.1680,0.0000
EC00287=7.9465,0.0000
EC00288=7.8844,0.0000
EC00289=7.7630,0.0000
EC00290=7.6803,0.0000
EC00291=7.7585,0.0000
EC00292=9.4604,0.0000
EC00293=12.4636,0.0000
EC00294=16.2505,0.0000
EC00295=20.3860,0.0000
EC00296=24.6140,0.0000
EC00297=28.7498,0.0000
EC00298=32.5363,0.0000
EC00299=35.5394,0.0000
EC00300=37.2413,0.0000
EC00301=37.3191,0.0000
EC00302=37.2369,0.0000
EC00303=37.1159,0.0000
EC00304=37.0536,0.0000
EC00305=37.8325,0.0000
EC00306=40.8660,0.0000
EC00307=43.3290,0.0000
EC00308=45.0000,0.0000
EC00309=46.6710,0.0000
EC00310=49.1340,0.0000
EC00311=52.1675,0.0000
EC00312=52.9464,0.0000
EC00313=52.8841,0.0000
EC00314=52.7631,0.0000
EC00315=52.6809,0.0000
EC00316=52.7587,0.0000
EC00317=54.4606,0.0000
EC00318=57.4637,0.0000
EC00319=61.2502,0.0000
EC00320=65.3860,0.0000
EC00321=69.6140,0.0000
EC00322=73.7495,0.0000
EC00323=77.5364,0.0000
EC00324=80.5396,0.0000
EC00325=82.2415,0.0000
EC00326=82.3197,0.0000
EC00327=82.2370,0.0000
EC00328=82.1156,0.0000
EC00329=82.0535,0.0000
EC00330=82.8320,0.0000
EC00331=85.8661,0.0000
EC00332=88.3294,0.0000
EC00333=90.0000,0.0000
EC00334=91.6706,0.0000
EC00335=94.1349,0.0000
EC00336=97.1678,0.0000
EC00337=97.9465,0.0000
EC00338=97.8844,0.0000
EC00339=97.7630,0.0000
EC00340=97.6803,0.0000
EC00341=97.7585,0.0000
EC00342=99.4604,0.0000
EC00343=102.4636,0.0000
EC00344=106.2505,0.0000
EC00345=110.3860,0.0000
EC00346=114.6140,0.0000
EC00347=118.7498,0.0000
EC00348=122.5363,0.0000
EC00349=125.5394,0.0000
EC00350=127.2413,0.0000
EC00351=127.3191,0.0000
EC00352=127.2369,0.0000
EC00353=127.1159,0.0000
EC00354=127.0536,0.0000
EC00355=127.8325,0.0000
EC00356=130.8660,0.0000
EC00357=133.3290,0.0000
EC00358=135.0000,0.0000
EC00359=136.6710,0.0000
EC00360=139.1340,0.0000
EC00361=142.1675,0.0000
EC00362=142.9464,0.0000
EC00363=142.8841,0.0000
EC00364=142.7631,0.0000
EC00365=142.6809,0.0000
EC00366=142.7587,0.0000
EC00367=144.4606,0.0000
EC00368=147.4637,0.0000
EC00369=151.2502,0.0000
EC00370=155.3860,0.0000
EC00371=159.6140,0.0000
EC00372=163.7495,0.0000
EC00373=167.5364,0.0000
EC00374=170.5396,0.0000
EC00375=172.2415,0.0000
EC00376=172.3197,0.0000
EC00377=172.2370,0.0000
EC00378=172.1156,0.0000
EC00379=172.0535,0.0000
EC00380=172.8320,0.0000
EC00381=175.8661,0.0000
EC00382=178.3294,0.0000
EC00383=180.0000,0.0000
EC00384=180.0000,0.0000
EC00385=-178.3294,0.0000
EC00386=-175.8651,0.0000
EC00387=-172.8322,0.0000
EC00388=-172.0535,0.0000
EC00389=-172.1156,0.0000
EC00390=-172.2370,0.0000
EC00391=-172.3197,0.0000
EC00392=-172.2415,0.0000
EC00393=-170.5396,0.0000
EC00394=-167.5364,0.0000
EC00395=-163.7495,0.0000
EC00396=-159.6140,0.0000
EC00397=-155.3860,0.0000
EC00398=-151.2502,0.0000
EC00399=-147.4637,0.0000
EC00400=-144.4606,0.0000
EC00401=-142.7587,0.0000
EC00402=-142.6809,0.0000
EC00403=-142.7631,0.0000
EC00404=-142.8841,0.0000
EC00405=-142.9464,0.0000
EC00406=-142.1675,0.0000
EC00407=-139.1340,0.0000
EC00408=-136.6710,0.0000
EC00409=-135.0000,0.0000
EC00410=-133.3290,0.0000
EC00411=-130.8660,0.0000
EC00412=-127.8325,0.0000
EC00413=-127.0536,0.0000
EC00414=-127.1159,0.0000
EC00415=-127.2369,0.0000
EC00416=-127.3191,0.0000
EC00417=-127.2413,0.0000
EC00418=-125.5394,0.0000
EC00419=-122.5363,0.0000
EC00420=-118.7498,0.0000
EC00421=-114.6140,0.0000
EC00422=-110.3860,0.0000
EC00423=-106.2505,0.0000
EC00424=-102.4636,0.0000
EC00425=-99.4604,0.0000
EC00426=-97.7585,0.0000
EC00427=-97.6803,0.0000
EC00428=-97.7630,0.0000
EC00429=-97.8844,0.0000
EC00430=-97.9465,0.0000
EC00431=-97.1680,0.0000
EC00432=-94.1339,0.0000
EC00433=-91.6706,0.0000
EC00434=-90.0000,0.0000
EC00435=-88.3294,0.0000
EC00436=-85.8651,0.0000
EC00437=-82.8322,0.0000
EC00438=-82.0535,0.0000
EC00439=-82.1156,0.0000
EC00440=-82.2370,0.0000
EC00441=-82.3197,0.0000
EC00442=-82.2415,0.0000
EC00443=-80.5396,0.0000
EC00444=-77.5364,0.0000
EC00445=-73.7495,0.0000
EC00446=-69.6140,0.0000
EC00447=-65.3860,0.0000
EC00448=-61.2502,0.0000
EC00449=-57.4637,0.0000
EC00450=-54.4606,0.0000
EC00451=-52.7587,0.0000
EC00452=-52.6809,0.0000
EC00453=-52.7631,0.0000
EC00454=-52.8841,0.0000
EC00455=-52.9464,0.0000
EC00456=-52.1675,0.0000
EC00457=-49.1340,0.0000
EC00458=-46.6710,0.0000
EC00459=-45.0000,0.0000
EC00460=-43.3290,0.0000
EC00461=-40.8660,0.0000
EC00462=-37.8325,0.0000
EC00463=-37.0536,0.0000
EC00464=-37.1159,0.0000
EC00465=-37.2369,0.0000
EC00466=-37.3191,0.0000
EC00467=-37.2413,0.0000
EC00468=-35.5394,0.0000
EC00469=-32.5363,0.0000
EC00470=-28.7498,0.0000
EC00471=-24.6140,0.0000
EC00472=-20.3860,0.0000
EC00473=-16.2505,0.0000
EC00474=-12.4636,0.0000
EC00475=-9.4604,0.0000
EC00476=-7.7585,0.0000
EC00477=-7.6803,0.0000
EC00478=-7.7630,0.0000
EC00479=-7.8844,0.0000
EC00480=-7.9465,0.0000
EC00481=-7.1678,0.0000
EC00482=-4.1349,0.0000
EC00483=-1.6706,0.0000
EC00484=0.0000,0.0000
EC00485=0.0000,0.0000
EC00486=1.6025,0.0000
EC00487=4.0449,0.0000
EC00488=7.0981,0.0000
EC00489=7.8538,0.0000
EC00490=7.7815,0.0000
EC00491=7.6711,0.0000
EC00492=7.6022,0.0000
EC00493=7.6844,0.0000
EC00494=9.3971,0.0000
EC00495=12.4165,0.0000
EC00496=16.2223,0.0000
EC00497=20.3773,0.0000
EC00498=24.6227,0.0000
EC00499=28.7775,0.0000
EC00500=32.5833,0.0000
EC00501=35.6027,0.0000
EC00502=37.3159,0.0000
EC00503=37.3980,0.0000
EC00504=37.3291,0.0000
EC00505=37.2193,0.0000
EC00506=37.1468,0.0000
EC00507=37.9017,0.0000
EC00508=40.9551,0.0000
EC00509=43.3970,0.0000
EC00510=45.0000,0.0000
EC00511=46.6030,0.0000
EC00512=49.0449,0.0000
EC00513=52.0983,0.0000
EC00514=52.8532,0.0000
EC00515=52.7807,0.0000
EC00516=52.6709,0.0000
EC00517=52.6020,0.0000
EC00518=52.6841,0.0000
EC00519=54.3973,0.0000
EC00520=57.4167,0.0000
EC00521=61.2225,0.0000
EC00522=65.3773,0.0000
EC00523=69.6227,0.0000
EC00524=73.7777,0.0000
EC00525=77.5835,0.0000
EC00526=80.6029,0.0000
EC00527=82.3156,0.0000
EC00528=82.3978,0.0000
EC00529=82.3289,0.0000
EC00530=82.2185,0.0000
EC00531=82.1462,0.0000
EC00532=82.9019,0.0000
EC00533=85.9551,0.0000
EC00534=88.3975,0.0000
EC00535=90.0000,0.0000
EC00536=91.6025,0.0000
EC00537=94.0449,0.0000
EC00538=97.0981,0.0000
EC00539=97.8538,0.0000
EC00540=97.7815,0.0000
EC00541=97.6711,0.0000
EC00542=97.6022,0.0000
EC00543=97.6844,0.0000
EC00544=99.3971,0.0000
EC00545=102.4165,0.0000
EC00546=106.2223,0.0000
EC00547=110.3773,0.0000
EC00548=114.6227,0.0000
EC00549=118.7775,0.0000
EC00550=122.5833,0.0000
EC00551=125.6027,0.0000
EC00552=127.3159,0.0000
EC00553=127.3980,0.0000
EC00554=127.3291,0.0000
EC00555=127.2193,0.0000
EC00556=127.1468,0.0000
EC00557=127.9017,0.0000
EC00558=130.9551,0.0000
EC00559=133.3970,0.0000
EC00560=135.0000,0.0000
EC00561=136.6030,0.0000
EC00562=139.0449,0.0000
EC00563=142.0983,0.0000
EC00564=142.8532,0.0000
EC00565=142.7807,0.0000
EC00566=142.6709,0.0000
EC00567=142.6020,0.0000
EC00568=142.6841,0.0000
EC00569=144.3973,0.0000
EC00570=147.4167,0.0000
EC00571=151.2225,0.0000
EC00572=155.3773,0.0000
EC00573=159.6227,0.0000
EC00574=163.7777,0.0000
EC00575=167.5835,0.0000
EC00576=170.6029,0.0000
EC00577=172.3156,0.0000
EC00578=172.3978,0.0000
EC00579=172.3289,0.0000
EC00580=172.2185,0.0000
EC00581=172.1462,0.0000
EC00582=172.9019,0.0000
EC00583=175.9551,0.0000
EC00584=178.3975,0.0000
EC00585=180.0000,0.0000
EC00586=180.0000,0.0000
EC00587=-178.3975,0.0000
EC00588=-175.9551,0.0000
EC00589=-172.9019,0.0000
EC00590=-172.1462,0.0000
EC00591=-172.2185,0.0000
EC00592=-172.3289,0.0000
EC00593=-172.3978,0.0000
EC00594=-172.3156,0.0000
EC00595=-170.6029,0.0000
EC00596=-167.5835,0.0000
EC00597=-163.7777,0.0000
EC00598=-159.6227,0.0000
EC00599=-155.3773,0.0000
EC00600=-151.2225,0.0000
EC00601=-147.4167,0.0000
EC00602=-144.3973,0.0000
EC00603=-142.6841,0.0000
EC00604=-142.6020,0.0000
EC00605=-142.6709,0.0000
EC00606=-142.7807,0.0000
EC00607=-142.8532,0.0000
EC00608=-142.0983,0.0000
EC00609=-139.0449,0.0000
EC00610=-136.6030,0.0000
EC00611=-135.0000,0.0000
EC00612=-133.3970,0.0000
EC00613=-130.9551,0.0000
EC00614=-127.9017,0.0000
EC00615=-127.1468,0.0000
EC00616=-127.2193,0.0000
EC00617=-127.3291,0.0000
EC00618=-127.3980,0.0000
EC00619=-127.3159,0.0000
EC00620=-125.6027,0.0000
EC00621=-122.5833,0.0000
EC00622=-118.7775,0.0000
EC00623=-114.6227,0.0000
EC00624=-110.3773,0.0000
EC00625=-106.2223,0.0000
EC00626=-102.4165,0.0000
EC00627=-99.3971,0.0000
EC00628=-97.6844,0.0000
EC00629=-97.6022,0.0000
EC00630=-97.6711,0.0000
EC00631=-97.7815,0.0000
EC00632=-97.8538,0.0000
EC00633=-97.0981,0.0000
EC00634=-94.0449,0.0000
EC00635=-91.6025,0.0000
EC00636=-90.0000,0.0000
EC00637=-88.3975,0.0000
EC00638=-85.9551,0.0000
EC00639=-82.9019,0.0000
EC00640=-82.1462,0.0000
EC00641=-82.2185,0.0000
EC00642=-82.3289,0.0000
EC00643=-82.3978,0.0000
EC00644=-82.3156,0.0000
EC00645=-80.6029,0.0000
EC00646=-77.5835,0.0000
EC00647=-73.7777,0.0000
EC00648=-69.6227,0.0000
EC00649=-65.3773,0.0000
EC00650=-61.2225,0.0000
EC00651=-57.4167,0.0000
EC00652=-54.3973,0.0000
EC00653=-52.6841,0.0000
EC00654=-52.6020,0.0000
EC00655=-52.6709,0.0000
EC00656=-52.7807,0.0000
EC00657=-52.8532,0.0000
EC00658=-52.0983,0.0000
EC00659=-49.0449,0.0000
EC00660=-46.6030,0.0000
EC00661=-45.0000,0.0000
EC00662=-43.3970,0.0000
EC00663=-40.9551,0.0000
EC00664=-37.9017,0.0000
EC00665=-37.1468,0.0000
EC00666=-37.2193,0.0000
EC00667=-37.3291,0.0000
EC00668=-37.3980,0.0000
EC00669=-37.3159,0.0000
EC00670=-35.6027,0.0000
EC00671=-32.5833,0.0000
EC00672=-28.7775,0.0000
EC00673=-24.6227,0.0000
EC00674=-20.3773,0.0000
EC00675=-16.2223,0.0000
EC00676=-12.4165,0.0000
EC00677=-9.3971,0.0000
EC00678=-7.6844,0.0000
EC00679=-7.6022,0.0000
EC00680=-7.6711,0.0000
EC00681=-7.7815,0.0000
EC00682=-7.8538,0.0000
EC00683=-7.0981,0.0000
EC00684=-4.0449,0.0000
EC00685=-1.6025,0.0000
EC00686=0.0000,0.0000
EC00687=0.0000,0.0000
EC00688=1.5376,0.0000
EC00689=3.9586,0.0000
EC00690=7.0327,0.0000
EC00691=7.7683,0.0000
EC00692=7.6919,0.0000
EC00693=7.5966,0.0000
EC00694=7.5446,0.0000
EC00695=7.6343,0.0000
EC00696=9.3569,0.0000
EC00697=12.3884,0.0000
EC00698=16.2065,0.0000
EC00699=20.3718,0.0000
EC00700=24.6278,0.0000
EC00701=28.7938,0.0000
EC00702=32.6119,0.0000
EC00703=35.6434,0.0000
EC00704=37.3659,0.0000
EC00705=37.4553,0.0000
EC00706=37.4027,0.0000
EC00707=37.3085,0.0000
EC00708=37.2322,0.0000
EC00709=37.9674,0.0000
EC00710=41.0417,0.0000
EC00711=43.4634,0.0000
EC00712=45.0000,0.0000
EC00713=46.5366,0.0000
EC00714=48.9583,0.0000
EC00715=52.0326,0.0000
EC00716=52.7678,0.0000
EC00717=52.6915,0.0000
EC00718=52.5973,0.0000
EC00719=52.5447,0.0000
EC00720=52.6341,0.0000
EC00721=54.3566,0.0000
EC00722=57.3881,0.0000
EC00723=61.2062,0.0000
EC00724=65.3722,0.0000
EC00725=69.6282,0.0000
EC00726=73.7935,0.0000
EC00727=77.6116,0.0000
EC00728=80.6431,0.0000
EC00729=82.3657,0.0000
EC00730=82.4554,0.0000
EC00731=82.4034,0.0000
EC00732=82.3081,0.0000
EC00733=82.2317,0.0000
EC00734=82.9673,0.0000
EC00735=86.0414,0.0000
EC00736=88.4624,0.0000
EC00737=90.0000,0.0000
EC00738=91.5365,0.0000
EC00739=93.9586,0.0000
EC00740=97.0327,0.0000
EC00741=97.7683,0.0000
EC00742=97.6919,0.0000
EC00743=97.5966,0.0000
EC00744=97.5446,0.0000
EC00745=97.6343,0.0000
EC00746=99.3569,0.0000
EC00747=102.3884,0.0000
EC00748=106.2065,0.0000
EC00749=110.3718,0.0000
EC00750=114.6278,0.0000
EC00751=118.7938,0.0000
EC00752=122.6119,0.0000
EC00753=125.6434,0.0000
EC00754=127.3659,0.0000
EC00755=127.4553,0.0000
EC00756=127.4027,0.0000
EC00757=127.3085,0.0000
EC00758=127.2322,0.0000
EC00759=127.9674,0.0000
EC00760=131.0417,0.0000
EC00761=133.4634,0.0000
EC00762=135.0000,0.0000
EC00763=136.5366,0.0000
EC00764=138.9583,0.0000
EC00765=142.0326,0.0000
EC00766=142.7678,0.0000
EC00767=142.6915,0.0000
EC00768=142.5973,0.0000
EC00769=142.5447,0.0000
EC00770=142.6341,0.0000
EC00771=144.3566,0.0000
EC00772=147.3881,0.0000
EC00773=151.2062,0.0000
EC00774=155.3722,0.0000
EC00775=159.6282,0.0000
EC00776=163.7935,0.0000
EC00777=167.6116,0.0000
EC00778=170.6431,0.0000
EC00779=172.3657,0.0000
EC00780=172.4554,0.0000
EC00781=172.4034,0.0000
EC00782=172.3081,0.0000
EC00783=172.2317,0.0000
EC00784=172.9673,0.0000
EC00785=176.0414,0.0000
EC00786=178.4624,0.0000
EC00787=180.0000,0.0000
EC00788=180.0000,0.0000
EC00789=-178.4635,0.0000
EC00790=-176.0414,0.0000
EC00791=-172.9673,0.0000
EC00792=-172.2317,0.0000
EC00793=-172.3081,0.0000
EC00794=-172.4034,0.0000
EC00795=-172.4554,0.0000
EC00796=-172.3657,0.0000
EC00797=-170.6431,0.0000
EC00798=-167.6116,0.0000
EC00799=-163.7935,0.0000
EC00800=-159.6282,0.0000
EC00801=-155.3722,0.0000
EC00802=-151.2062,0.0000
EC00803=-147.3881,0.0000
EC00804=-144.3566,0.0000
EC00805=-142.6341,0.0000
EC00806=-142.5447,0.0000
EC00807=-142.5973,0.0000
EC00808=-142.6915,0.0000
EC00809=-142.7678,0.0000
EC00810=-142.0326,0.0000
